LIN {X 0,Y 367.763,Z 472.156,A -85,B 0,C 180,E1 -12598.905,E2 -12598.905} C_VEL
LIN {X 0,Y 367.872,Z 472.925,A -85,B 0,C 180,E1 -12601.095,E2 -12601.095} C_VEL
LIN {X 0,Y 368.13,Z 472.594,A -85,B 0,C 180,E1 -12603.283,E2 -12603.283} C_VEL
LIN {X 0,Y 368.318,Z 471.288,A -85,B 0,C 180,E1 -12605.475,E2 -12605.475} C_VEL
LIN {X 0,Y 368.311,Z 470.292,A -85,B 0,C 180,E1 -12606.574,E2 -12606.574} C_VEL
LIN {X 0,Y 368.949,Z 467.35,A -85,B 0,C 180,E1 -12608.765,E2 -12608.765} C_VEL
LIN {X 0,Y 369.704,Z 463.365,A -85,B 0,C 180,E1 -12610.958,E2 -12610.958} C_VEL
LIN {X 0,Y 370.548,Z 458.282,A -85,B 0,C 180,E1 -12613.156,E2 -12613.156} C_VEL
LIN {X 0,Y 371.827,Z 451.616,A -85,B 0,C 180,E1 -12615.426,E2 -12615.426} C_VEL
LIN {X 0,Y 373.279,Z 444.114,A -85,B 0,C 180,E1 -12617.532,E2 -12617.532} C_VEL
LIN {X 0,Y 375.138,Z 434.807,A -85,B 0,C 180,E1 -12619.707,E2 -12619.707} C_VEL
LIN {X 0,Y 377.114,Z 425.21,A -85,B 0,C 180,E1 -12621.596,E2 -12621.596} C_VEL
LIN {X 0,Y 379.312,Z 413.922,A -85,B 0,C 180,E1 -12623.475,E2 -12623.475} C_VEL
LIN {X 0,Y 381.513,Z 402.619,A -85,B 0,C 180,E1 -12625.068,E2 -12625.068} C_VEL
LIN {X 0,Y 383.923,Z 389.529,A -85,B 0,C 180,E1 -12626.647,E2 -12626.647} C_VEL
LIN {X 0,Y 386.088,Z 376.887,A -85,B 0,C 180,E1 -12627.952,E2 -12627.952} C_VEL
LIN {X 0,Y 388.194,Z 363.605,A -85,B 0,C 180,E1 -12629.114,E2 -12629.114} C_VEL
LIN {X 0,Y 390.459,Z 347.831,A -85,B 0,C 180,E1 -12630.264,E2 -12630.264} C_VEL
LIN {X 0,Y 392.54,Z 330.694,A -85,B 0,C 180,E1 -12631.279,E2 -12631.279} C_VEL
LIN {X 0,Y 394.4,Z 312.888,A -85,B 0,C 180,E1 -12632.089,E2 -12632.089} C_VEL
LIN {X 0,Y 396.951,Z 285.614,A -85,B 0,C 180,E1 -12632.985,E2 -12632.985} C_VEL
LIN {X 0,Y 404.321,Z 221.247,A -85,B 0,C 180,E1 -12635.04,E2 -12635.04} C_VEL
LIN {X 0,Y 411.797,Z 167.375,A -85,B 0,C 180,E1 -12636.792,E2 -12636.792} C_VEL
LIN {X 0,Y 409.225,Z 162.785,A -85,B 0,C 180,E1 -12637.954,E2 -12637.954} C_VEL
LIN {X 0,Y 406.549,Z 158.694,A -85,B 0,C 180,E1 -12639.413,E2 -12639.413} C_VEL
LIN {X 0,Y 403.9,Z 155.628,A -85,B 0,C 180,E1 -12641.392,E2 -12641.392} C_VEL
LIN {X 0,Y 403.16,Z 154.958,A -85,B 0,C 180,E1 -12642.248,E2 -12642.248} C_VEL
LIN {X 0,Y 402.329,Z 154.997,A -85,B 0,C 180,E1 -12643.844,E2 -12643.844} C_VEL
LIN {X 0,Y 402.381,Z 156.776,A -85,B 0,C 180,E1 -12645.734,E2 -12645.734} C_VEL
LIN {X 0,Y 403.284,Z 159.225,A -85,B 0,C 180,E1 -12647.232,E2 -12647.232} C_VEL
LIN {X 0,Y 404.582,Z 162.984,A -85,B 0,C 180,E1 -12648.582,E2 -12648.582} C_VEL
LIN {X 0,Y 406.534,Z 167.981,A -85,B 0,C 180,E1 -12649.976,E2 -12649.976} C_VEL
LIN {X 0,Y 408.747,Z 174.299,A -85,B 0,C 180,E1 -12651.27,E2 -12651.27} C_VEL
LIN {X 0,Y 409.591,Z 177.225,A -85,B 0,C 180,E1 -12651.738,E2 -12651.738} C_VEL
LIN {X 0,Y 409.008,Z 196.365,A -85,B 0,C 180,E1 -12652.915,E2 -12652.915} C_VEL
LIN {X 0,Y 401.408,Z 257.244,A -85,B 0,C 180,E1 -12654.859,E2 -12654.859} C_VEL
LIN {X 0,Y 394.781,Z 323.074,A -85,B 0,C 180,E1 -12656.91,E2 -12656.91} C_VEL
LIN {X 0,Y 392.088,Z 351.319,A -85,B 0,C 180,E1 -12657.812,E2 -12657.812} C_VEL
LIN {X 0,Y 389.573,Z 370.272,A -85,B 0,C 180,E1 -12658.606,E2 -12658.606} C_VEL
LIN {X 0,Y 387.34,Z 385.034,A -85,B 0,C 180,E1 -12659.391,E2 -12659.391} C_VEL
LIN {X 0,Y 384.488,Z 402.958,A -85,B 0,C 180,E1 -12660.577,E2 -12660.577} C_VEL
LIN {X 0,Y 381.88,Z 418.792,A -85,B 0,C 180,E1 -12661.862,E2 -12661.862} C_VEL
LIN {X 0,Y 379.221,Z 433.932,A -85,B 0,C 180,E1 -12663.319,E2 -12663.319} C_VEL
LIN {X 0,Y 376.682,Z 448.794,A -85,B 0,C 180,E1 -12665.03,E2 -12665.03} C_VEL
LIN {X 0,Y 374.432,Z 462.363,A -85,B 0,C 180,E1 -12666.884,E2 -12666.884} C_VEL
LIN {X 0,Y 372.559,Z 473.762,A -85,B 0,C 180,E1 -12668.707,E2 -12668.707} C_VEL
LIN {X 0,Y 370.81,Z 485.557,A -85,B 0,C 180,E1 -12670.916,E2 -12670.916} C_VEL
LIN {X 0,Y 369.526,Z 495.557,A -85,B 0,C 180,E1 -12673.139,E2 -12673.139} C_VEL
LIN {X 0,Y 368.683,Z 503.018,A -85,B 0,C 180,E1 -12675.087,E2 -12675.087} C_VEL
LIN {X 0,Y 368.088,Z 510.152,A -85,B 0,C 180,E1 -12677.315,E2 -12677.315} C_VEL
LIN {X 0,Y 367.701,Z 516.033,A -85,B 0,C 180,E1 -12679.538,E2 -12679.538} C_VEL
LIN {X 0,Y 367.598,Z 520.659,A -85,B 0,C 180,E1 -12681.755,E2 -12681.755} C_VEL
LIN {X 0,Y 367.722,Z 523.703,A -85,B 0,C 180,E1 -12683.633,E2 -12683.633} C_VEL
LIN {X 0,Y 367.603,Z 525.957,A -85,B 0,C 180,E1 -12685.613,E2 -12685.613} C_VEL
LIN {X 0,Y 367.759,Z 527.494,A -85,B 0,C 180,E1 -12687.809,E2 -12687.809} C_VEL
LIN {X 0,Y 367.812,Z 527.835,A -85,B 0,C 180,E1 -12689.999,E2 -12689.999} C_VEL
LIN {X 0,Y 367.777,Z 527.091,A -85,B 0,C 180,E1 -12692.19,E2 -12692.19} C_VEL
LIN {X 0,Y 367.764,Z 526.32,A -85,B 0,C 180,E1 -12693.286,E2 -12693.286} C_VEL
LIN {X 0,Y 367.724,Z 523.809,A -85,B 0,C 180,E1 -12695.483,E2 -12695.483} C_VEL
LIN {X 0,Y 367.682,Z 520.167,A -85,B 0,C 180,E1 -12697.689,E2 -12697.689} C_VEL
LIN {X 0,Y 367.668,Z 515.275,A -85,B 0,C 180,E1 -12699.905,E2 -12699.905} C_VEL
LIN {X 0,Y 367.978,Z 509.03,A -85,B 0,C 180,E1 -12702.127,E2 -12702.127} C_VEL
LIN {X 0,Y 368.449,Z 501.363,A -85,B 0,C 180,E1 -12704.357,E2 -12704.357} C_VEL
LIN {X 0,Y 369.148,Z 493.386,A -85,B 0,C 180,E1 -12706.308,E2 -12706.308} C_VEL
LIN {X 0,Y 370.131,Z 483.052,A -85,B 0,C 180,E1 -12708.427,E2 -12708.427} C_VEL
LIN {X 0,Y 371.25,Z 472.812,A -85,B 0,C 180,E1 -12710.211,E2 -12710.211} C_VEL
LIN {X 0,Y 372.828,Z 459.757,A -85,B 0,C 180,E1 -12712.148,E2 -12712.148} C_VEL
LIN {X 0,Y 374.395,Z 446.566,A -85,B 0,C 180,E1 -12713.802,E2 -12713.802} C_VEL
LIN {X 0,Y 376.106,Z 432.348,A -85,B 0,C 180,E1 -12715.305,E2 -12715.305} C_VEL
LIN {X 0,Y 377.884,Z 416.601,A -85,B 0,C 180,E1 -12716.688,E2 -12716.688} C_VEL
LIN {X 0,Y 379.684,Z 400.106,A -85,B 0,C 180,E1 -12717.863,E2 -12717.863} C_VEL
LIN {X 0,Y 381.204,Z 383.748,A -85,B 0,C 180,E1 -12718.792,E2 -12718.792} C_VEL
LIN {X 0,Y 382.585,Z 366.326,A -85,B 0,C 180,E1 -12719.545,E2 -12719.545} C_VEL
LIN {X 0,Y 383.648,Z 349.415,A -85,B 0,C 180,E1 -12720.059,E2 -12720.059} C_VEL
LIN {X 0,Y 390.23,Z 192.191,A -85,B 0,C 180,E1 -12723.84,E2 -12723.84} C_VEL
LIN {X 0,Y 386.053,Z 158.999,A -85,B 0,C 180,E1 -12725.094,E2 -12725.094} C_VEL
LIN {X 0,Y 380.743,Z 146.981,A -85,B 0,C 180,E1 -12725.89,E2 -12725.89} C_VEL
LIN {X 0,Y 373.264,Z 123.838,A -85,B 0,C 180,E1 -12729.469,E2 -12729.469} C_VEL
LIN {X 0,Y 368.96,Z 110.84,A -85,B 0,C 180,E1 -12731.621,E2 -12731.621} C_VEL
LIN {X 0,Y 368.919,Z 110.844,A -85,B 0,C 180,E1 -12735.182,E2 -12735.182} C_VEL
LIN {X 0,Y 368.879,Z 110.849,A -85,B 0,C 180,E1 -12738.177,E2 -12738.177} C_VEL
LIN {X 0,Y 368.905,Z 110.841,A -85,B 0,C 180,E1 -12741.359,E2 -12741.359} C_VEL
LIN {X 0,Y 368.932,Z 110.838,A -85,B 0,C 180,E1 -12745.146,E2 -12745.146} C_VEL
LIN {X 0,Y 368.924,Z 110.839,A -85,B 0,C 180,E1 -12749.046,E2 -12749.046} C_VEL
LIN {X 0,Y 368.982,Z 110.833,A -85,B 0,C 180,E1 -12751.564,E2 -12751.564} C_VEL
LIN {X 0,Y 368.953,Z 110.836,A -85,B 0,C 180,E1 -12755.224,E2 -12755.224} C_VEL
LIN {X 0,Y 368.932,Z 110.838,A -85,B 0,C 180,E1 -12758.973,E2 -12758.973} C_VEL
LIN {X 0,Y 368.986,Z 110.834,A -85,B 0,C 180,E1 -12762.257,E2 -12762.257} C_VEL
LIN {X 0,Y 369.012,Z 110.832,A -85,B 0,C 180,E1 -12765.665,E2 -12765.665} C_VEL
LIN {X 0,Y 369.025,Z 110.827,A -85,B 0,C 180,E1 -12769.021,E2 -12769.021} C_VEL
LIN {X 0,Y 369.183,Z 110.808,A -85,B 0,C 180,E1 -12772.342,E2 -12772.342} C_VEL
LIN {X 0,Y 369.14,Z 110.812,A -85,B 0,C 180,E1 -12774.538,E2 -12774.538} C_VEL
LIN {X 0,Y 369.314,Z 110.795,A -85,B 0,C 180,E1 -12777.819,E2 -12777.819} C_VEL
LIN {X 0,Y 369.454,Z 110.776,A -85,B 0,C 180,E1 -12780,E2 -12780} C_VEL
LIN {X 0,Y 369.314,Z 110.792,A -85,B 0,C 180,E1 -12782.181,E2 -12782.181} C_VEL
LIN {X 0,Y 369.2,Z 110.805,A -85,B 0,C 180,E1 -12786.616,E2 -12786.616} C_VEL
LIN {X 0,Y 369.133,Z 110.814,A -85,B 0,C 180,E1 -12788.761,E2 -12788.761} C_VEL
LIN {X 0,Y 369.001,Z 110.83,A -85,B 0,C 180,E1 -12792.094,E2 -12792.094} C_VEL
LIN {X 0,Y 368.993,Z 110.836,A -85,B 0,C 180,E1 -12795.465,E2 -12795.465} C_VEL
LIN {X 0,Y 368.954,Z 110.838,A -85,B 0,C 180,E1 -12798.894,E2 -12798.894} C_VEL
LIN {X 0,Y 368.928,Z 110.839,A -85,B 0,C 180,E1 -12802.395,E2 -12802.395} C_VEL
LIN {X 0,Y 368.996,Z 110.83,A -85,B 0,C 180,E1 -12805.981,E2 -12805.981} C_VEL
LIN {X 0,Y 368.911,Z 110.842,A -85,B 0,C 180,E1 -12809.691,E2 -12809.691} C_VEL
LIN {X 0,Y 368.893,Z 110.85,A -85,B 0,C 180,E1 -12813.044,E2 -12813.044} C_VEL
LIN {X 0,Y 368.914,Z 110.841,A -85,B 0,C 180,E1 -12816.197,E2 -12816.197} C_VEL
LIN {X 0,Y 368.901,Z 110.849,A -85,B 0,C 180,E1 -12818.953,E2 -12818.953} C_VEL
LIN {X 0,Y 368.878,Z 110.845,A -85,B 0,C 180,E1 -12822.01,E2 -12822.01} C_VEL
LIN {X 0,Y 368.905,Z 110.844,A -85,B 0,C 180,E1 -12825.181,E2 -12825.181} C_VEL
LIN {X 0,Y 368.907,Z 110.842,A -85,B 0,C 180,E1 -12828.182,E2 -12828.182} C_VEL
LIN {X 0,Y 368.908,Z 110.842,A -85,B 0,C 180,E1 -12831.36,E2 -12831.36} C_VEL
LIN {X 0,Y 368.934,Z 110.84,A -85,B 0,C 180,E1 -12835.147,E2 -12835.147} C_VEL
LIN {X 0,Y 368.927,Z 110.841,A -85,B 0,C 180,E1 -12839.047,E2 -12839.047} C_VEL
LIN {X 0,Y 368.961,Z 110.838,A -85,B 0,C 180,E1 -12842.797,E2 -12842.797} C_VEL
LIN {X 0,Y 368.944,Z 110.839,A -85,B 0,C 180,E1 -12846.114,E2 -12846.114} C_VEL
LIN {X 0,Y 368.944,Z 110.839,A -85,B 0,C 180,E1 -12849.948,E2 -12849.948} C_VEL
LIN {X 0,Y 368.975,Z 110.833,A -85,B 0,C 180,E1 -12853.399,E2 -12853.399} C_VEL
LIN {X 0,Y 369.057,Z 110.824,A -85,B 0,C 180,E1 -12856.791,E2 -12856.791} C_VEL
LIN {X 0,Y 369.07,Z 110.826,A -85,B 0,C 180,E1 -12860.133,E2 -12860.133} C_VEL
LIN {X 0,Y 369.189,Z 110.811,A -85,B 0,C 180,E1 -12862.343,E2 -12862.343} C_VEL
LIN {X 0,Y 369.144,Z 110.814,A -85,B 0,C 180,E1 -12864.538,E2 -12864.538} C_VEL
LIN {X 0,Y 369.317,Z 110.794,A -85,B 0,C 180,E1 -12867.82,E2 -12867.82} C_VEL
LIN {X 0,Y 369.457,Z 110.779,A -85,B 0,C 180,E1 -12870.001,E2 -12870.001} C_VEL
LIN {X 0,Y 369.317,Z 110.795,A -85,B 0,C 180,E1 -12872.182,E2 -12872.182} C_VEL
LIN {X 0,Y 369.21,Z 110.805,A -85,B 0,C 180,E1 -12876.559,E2 -12876.559} C_VEL
LIN {X 0,Y 369.139,Z 110.812,A -85,B 0,C 180,E1 -12878.762,E2 -12878.762} C_VEL
LIN {X 0,Y 369.007,Z 110.833,A -85,B 0,C 180,E1 -12882.094,E2 -12882.094} C_VEL
LIN {X 0,Y 369,Z 110.833,A -85,B 0,C 180,E1 -12885.465,E2 -12885.465} C_VEL
LIN {X 0,Y 368.96,Z 110.835,A -85,B 0,C 180,E1 -12888.895,E2 -12888.895} C_VEL
LIN {X 0,Y 368.934,Z 110.838,A -85,B 0,C 180,E1 -12892.396,E2 -12892.396} C_VEL
LIN {X 0,Y 369.002,Z 110.832,A -85,B 0,C 180,E1 -12895.981,E2 -12895.981} C_VEL
LIN {X 0,Y 368.917,Z 110.845,A -85,B 0,C 180,E1 -12899.691,E2 -12899.691} C_VEL
LIN {X 0,Y 368.899,Z 110.844,A -85,B 0,C 180,E1 -12903.044,E2 -12903.044} C_VEL
LIN {X 0,Y 368.92,Z 110.84,A -85,B 0,C 180,E1 -12906.197,E2 -12906.197} C_VEL
LIN {X 0,Y 368.906,Z 110.844,A -85,B 0,C 180,E1 -12908.954,E2 -12908.954} C_VEL
LIN {X 0,Y 368.885,Z 110.845,A -85,B 0,C 180,E1 -12912.01,E2 -12912.01} C_VEL
LIN {X 0,Y 368.885,Z 110.846,A -85,B 0,C 180,E1 -12914.768,E2 -12914.768} C_VEL
LIN {X 0,Y 368.259,Z 110.929,A -85,B 0,C 180,E1 -12915.679,E2 -12915.679} C_VEL
LIN {X 0,Y 365.4,Z 111.29,A -85,B 0,C 180,E1 -12917.16,E2 -12917.16} C_VEL
LIN {X 0,Y 362.957,Z 111.592,A -85,B 0,C 180,E1 -12918.358,E2 -12918.358} C_VEL
LIN {X 0,Y 361.915,Z 111.718,A -85,B 0,C 180,E1 -12919.286,E2 -12919.286} C_VEL
LIN {X 0,Y 361.836,Z 111.724,A -85,B 0,C 180,E1 -12919.6,E2 -12919.6} C_VEL
LIN {X 0,Y 361.894,Z 111.804,A -85,B 0,C 180,E1 -12923.315,E2 -12923.315} C_VEL
LIN {X 0,Y 362.879,Z 114.579,A -85,B 0,C 180,E1 -12923.489,E2 -12923.489} C_VEL
LIN {X 0,Y 375.869,Z 139.954,A -85,B 0,C 180,E1 -12925.358,E2 -12925.358} C_VEL
LIN {X 0,Y 383.362,Z 155.105,A -85,B 0,C 180,E1 -12926.389,E2 -12926.389} C_VEL
LIN {X 0,Y 377.045,Z 300.554,A -85,B 0,C 180,E1 -12929.976,E2 -12929.976} C_VEL
LIN {X 0,Y 376.115,Z 317.935,A -85,B 0,C 180,E1 -12930.626,E2 -12930.626} C_VEL
LIN {X 0,Y 374.874,Z 335.248,A -85,B 0,C 180,E1 -12931.502,E2 -12931.502} C_VEL
LIN {X 0,Y 373.524,Z 351.415,A -85,B 0,C 180,E1 -12932.55,E2 -12932.55} C_VEL
LIN {X 0,Y 371.952,Z 367.033,A -85,B 0,C 180,E1 -12933.79,E2 -12933.79} C_VEL
LIN {X 0,Y 370.293,Z 381.51,A -85,B 0,C 180,E1 -12935.17,E2 -12935.17} C_VEL
LIN {X 0,Y 368.602,Z 396.146,A -85,B 0,C 180,E1 -12936.843,E2 -12936.843} C_VEL
LIN {X 0,Y 367.227,Z 407.642,A -85,B 0,C 180,E1 -12938.383,E2 -12938.383} C_VEL
LIN {X 0,Y 365.713,Z 420.041,A -85,B 0,C 180,E1 -12940.331,E2 -12940.331} C_VEL
LIN {X 0,Y 364.399,Z 430.687,A -85,B 0,C 180,E1 -12942.316,E2 -12942.316} C_VEL
LIN {X 0,Y 363.327,Z 439.7,A -85,B 0,C 180,E1 -12944.288,E2 -12944.288} C_VEL
LIN {X 0,Y 362.42,Z 448.408,A -85,B 0,C 180,E1 -12946.544,E2 -12946.544} C_VEL
LIN {X 0,Y 361.695,Z 455.627,A -85,B 0,C 180,E1 -12948.796,E2 -12948.796} C_VEL
LIN {X 0,Y 361.288,Z 461.435,A -85,B 0,C 180,E1 -12951.047,E2 -12951.047} C_VEL
LIN {X 0,Y 361.011,Z 466.025,A -85,B 0,C 180,E1 -12953.292,E2 -12953.292} C_VEL
LIN {X 0,Y 360.792,Z 469.537,A -85,B 0,C 180,E1 -12955.531,E2 -12955.531} C_VEL
LIN {X 0,Y 360.773,Z 471.872,A -85,B 0,C 180,E1 -12957.767,E2 -12957.767} C_VEL
LIN {X 0,Y 360.743,Z 473.22,A -85,B 0,C 180,E1 -12960,E2 -12960} C_VEL
LIN {X 0,Y 360.957,Z 473.516,A -85,B 0,C 180,E1 -12962.232,E2 -12962.232} C_VEL
LIN {X 0,Y 361.142,Z 472.773,A -85,B 0,C 180,E1 -12964.464,E2 -12964.464} C_VEL
LIN {X 0,Y 361.296,Z 471.082,A -85,B 0,C 180,E1 -12966.702,E2 -12966.702} C_VEL
LIN {X 0,Y 361.982,Z 468.215,A -85,B 0,C 180,E1 -12968.935,E2 -12968.935} C_VEL
LIN {X 0,Y 362.787,Z 464.338,A -85,B 0,C 180,E1 -12971.17,E2 -12971.17} C_VEL
LIN {X 0,Y 363.683,Z 459.323,A -85,B 0,C 180,E1 -12973.408,E2 -12973.408} C_VEL
LIN {X 0,Y 365.063,Z 452.768,A -85,B 0,C 180,E1 -12975.723,E2 -12975.723} C_VEL
LIN {X 0,Y 366.634,Z 445.41,A -85,B 0,C 180,E1 -12977.861,E2 -12977.861} C_VEL
LIN {X 0,Y 368.616,Z 436.268,A -85,B 0,C 180,E1 -12980.071,E2 -12980.071} C_VEL
LIN {X 0,Y 371.062,Z 425.321,A -85,B 0,C 180,E1 -12982.259,E2 -12982.259} C_VEL
LIN {X 0,Y 373.402,Z 414.056,A -85,B 0,C 180,E1 -12984.165,E2 -12984.165} C_VEL
LIN {X 0,Y 375.766,Z 402.839,A -85,B 0,C 180,E1 -12985.757,E2 -12985.757} C_VEL
LIN {X 0,Y 378.539,Z 388.47,A -85,B 0,C 180,E1 -12987.505,E2 -12987.505} C_VEL
LIN {X 0,Y 381.359,Z 372.824,A -85,B 0,C 180,E1 -12989.082,E2 -12989.082} C_VEL
LIN {X 0,Y 384.215,Z 355.813,A -85,B 0,C 180,E1 -12990.474,E2 -12990.474} C_VEL
LIN {X 0,Y 386.746,Z 338.182,A -85,B 0,C 180,E1 -12991.634,E2 -12991.634} C_VEL
LIN {X 0,Y 388.751,Z 321.708,A -85,B 0,C 180,E1 -12992.498,E2 -12992.498} C_VEL
LIN {X 0,Y 390.581,Z 303.73,A -85,B 0,C 180,E1 -12993.208,E2 -12993.208} C_VEL
LIN {X 0,Y 397.716,Z 242.686,A -85,B 0,C 180,E1 -12995.198,E2 -12995.198} C_VEL
LIN {X 0,Y 408.086,Z 171.591,A -85,B 0,C 180,E1 -12997.562,E2 -12997.562} C_VEL
LIN {X 0,Y 406.02,Z 168.026,A -85,B 0,C 180,E1 -12998.612,E2 -12998.612} C_VEL
LIN {X 0,Y 404.236,Z 165.141,A -85,B 0,C 180,E1 -12999.709,E2 -12999.709} C_VEL
LIN {X 0,Y 402.038,Z 162.435,A -85,B 0,C 180,E1 -13001.503,E2 -13001.503} C_VEL
LIN {X 0,Y 401.149,Z 161.75,A -85,B 0,C 180,E1 -13002.622,E2 -13002.622} C_VEL
LIN {X 0,Y 400.531,Z 162.015,A -85,B 0,C 180,E1 -13003.993,E2 -13003.993} C_VEL
LIN {X 0,Y 400.659,Z 163.827,A -85,B 0,C 180,E1 -13005.822,E2 -13005.822} C_VEL
LIN {X 0,Y 401.583,Z 166.692,A -85,B 0,C 180,E1 -13007.371,E2 -13007.371} C_VEL
LIN {X 0,Y 403.632,Z 172.828,A -85,B 0,C 180,E1 -13009.313,E2 -13009.313} C_VEL
LIN {X 0,Y 405.733,Z 179.636,A -85,B 0,C 180,E1 -13010.767,E2 -13010.767} C_VEL
LIN {X 0,Y 406.152,Z 181.286,A -85,B 0,C 180,E1 -13011.038,E2 -13011.038} C_VEL
LIN {X 0,Y 405.317,Z 198.198,A -85,B 0,C 180,E1 -13012.103,E2 -13012.103} C_VEL
LIN {X 0,Y 396.177,Z 266.329,A -85,B 0,C 180,E1 -13014.324,E2 -13014.324} C_VEL
LIN {X 0,Y 389.101,Z 332.133,A -85,B 0,C 180,E1 -13016.424,E2 -13016.424} C_VEL
LIN {X 0,Y 386.846,Z 352.633,A -85,B 0,C 180,E1 -13017.128,E2 -13017.128} C_VEL
LIN {X 0,Y 384.101,Z 371.38,A -85,B 0,C 180,E1 -13017.952,E2 -13017.952} C_VEL
LIN {X 0,Y 381.631,Z 386.548,A -85,B 0,C 180,E1 -13018.805,E2 -13018.805} C_VEL
LIN {X 0,Y 378.451,Z 404.704,A -85,B 0,C 180,E1 -13020.06,E2 -13020.06} C_VEL
LIN {X 0,Y 375.719,Z 419.977,A -85,B 0,C 180,E1 -13021.358,E2 -13021.358} C_VEL
LIN {X 0,Y 372.732,Z 435.816,A -85,B 0,C 180,E1 -13022.958,E2 -13022.958} C_VEL
LIN {X 0,Y 370.057,Z 450.273,A -85,B 0,C 180,E1 -13024.702,E2 -13024.702} C_VEL
LIN {X 0,Y 367.778,Z 463.128,A -85,B 0,C 180,E1 -13026.527,E2 -13026.527} C_VEL
LIN {X 0,Y 365.886,Z 473.862,A -85,B 0,C 180,E1 -13028.299,E2 -13028.299} C_VEL
LIN {X 0,Y 364.173,Z 484.144,A -85,B 0,C 180,E1 -13030.261,E2 -13030.261} C_VEL
LIN {X 0,Y 362.743,Z 494.248,A -85,B 0,C 180,E1 -13032.523,E2 -13032.523} C_VEL
LIN {X 0,Y 361.685,Z 502.788,A -85,B 0,C 180,E1 -13034.791,E2 -13034.791} C_VEL
LIN {X 0,Y 361.047,Z 510.035,A -85,B 0,C 180,E1 -13037.134,E2 -13037.134} C_VEL
LIN {X 0,Y 360.623,Z 515.639,A -85,B 0,C 180,E1 -13039.33,E2 -13039.33} C_VEL
LIN {X 0,Y 360.519,Z 520.243,A -85,B 0,C 180,E1 -13041.592,E2 -13041.592} C_VEL
LIN {X 0,Y 360.644,Z 523.385,A -85,B 0,C 180,E1 -13043.642,E2 -13043.642} C_VEL
LIN {X 0,Y 360.532,Z 525.452,A -85,B 0,C 180,E1 -13045.527,E2 -13045.527} C_VEL
LIN {X 0,Y 360.691,Z 526.924,A -85,B 0,C 180,E1 -13047.766,E2 -13047.766} C_VEL
LIN {X 0,Y 360.765,Z 527.242,A -85,B 0,C 180,E1 -13049.999,E2 -13049.999} C_VEL
LIN {X 0,Y 360.711,Z 526.425,A -85,B 0,C 180,E1 -13052.232,E2 -13052.232} C_VEL
LIN {X 0,Y 360.557,Z 524.488,A -85,B 0,C 180,E1 -13054.471,E2 -13054.471} C_VEL
LIN {X 0,Y 360.695,Z 521.812,A -85,B 0,C 180,E1 -13056.43,E2 -13056.43} C_VEL
LIN {X 0,Y 360.595,Z 517.008,A -85,B 0,C 180,E1 -13058.969,E2 -13058.969} C_VEL
LIN {X 0,Y 360.754,Z 511.368,A -85,B 0,C 180,E1 -13061.233,E2 -13061.233} C_VEL
LIN {X 0,Y 361.178,Z 504.313,A -85,B 0,C 180,E1 -13063.503,E2 -13063.503} C_VEL
LIN {X 0,Y 361.821,Z 495.725,A -85,B 0,C 180,E1 -13065.779,E2 -13065.779} C_VEL
LIN {X 0,Y 362.713,Z 486.824,A -85,B 0,C 180,E1 -13067.768,E2 -13067.768} C_VEL
LIN {X 0,Y 363.81,Z 476.313,A -85,B 0,C 180,E1 -13069.758,E2 -13069.758} C_VEL
LIN {X 0,Y 365.307,Z 463.947,A -85,B 0,C 180,E1 -13071.736,E2 -13071.736} C_VEL
LIN {X 0,Y 366.89,Z 451.226,A -85,B 0,C 180,E1 -13073.458,E2 -13073.458} C_VEL
LIN {X 0,Y 368.615,Z 436.88,A -85,B 0,C 180,E1 -13075.1,E2 -13075.1} C_VEL
LIN {X 0,Y 370.387,Z 422.46,A -85,B 0,C 180,E1 -13076.48,E2 -13076.48} C_VEL
LIN {X 0,Y 372.178,Z 406.983,A -85,B 0,C 180,E1 -13077.709,E2 -13077.709} C_VEL
LIN {X 0,Y 373.777,Z 391.291,A -85,B 0,C 180,E1 -13078.727,E2 -13078.727} C_VEL
LIN {X 0,Y 375.357,Z 374.103,A -85,B 0,C 180,E1 -13079.592,E2 -13079.592} C_VEL
LIN {X 0,Y 376.663,Z 356.279,A -85,B 0,C 180,E1 -13080.25,E2 -13080.25} C_VEL
LIN {X 0,Y 383.889,Z 193.183,A -85,B 0,C 180,E1 -13084.298,E2 -13084.298} C_VEL
LIN {X 0,Y 379.923,Z 161.529,A -85,B 0,C 180,E1 -13085.518,E2 -13085.518} C_VEL
LIN {X 0,Y 373.298,Z 146.581,A -85,B 0,C 180,E1 -13086.519,E2 -13086.519} C_VEL
LIN {X 0,Y 367.039,Z 127.165,A -85,B 0,C 180,E1 -13089.578,E2 -13089.578} C_VEL
LIN {X 0,Y 361.894,Z 111.721,A -85,B 0,C 180,E1 -13092.17,E2 -13092.17} C_VEL
LIN {X 0,Y 361.842,Z 111.726,A -85,B 0,C 180,E1 -13095.636,E2 -13095.636} C_VEL
LIN {X 0,Y 361.831,Z 111.723,A -85,B 0,C 180,E1 -13099.244,E2 -13099.244} C_VEL
LIN {X 0,Y 361.867,Z 111.72,A -85,B 0,C 180,E1 -13102.775,E2 -13102.775} C_VEL
LIN {X 0,Y 361.851,Z 111.722,A -85,B 0,C 180,E1 -13105.72,E2 -13105.72} C_VEL
LIN {X 0,Y 361.872,Z 111.719,A -85,B 0,C 180,E1 -13109.672,E2 -13109.672} C_VEL
LIN {X 0,Y 361.95,Z 111.709,A -85,B 0,C 180,E1 -13113.475,E2 -13113.475} C_VEL
LIN {X 0,Y 361.885,Z 111.716,A -85,B 0,C 180,E1 -13117.145,E2 -13117.145} C_VEL
LIN {X 0,Y 361.916,Z 111.712,A -85,B 0,C 180,E1 -13120.724,E2 -13120.724} C_VEL
LIN {X 0,Y 361.944,Z 111.712,A -85,B 0,C 180,E1 -13124.226,E2 -13124.226} C_VEL
LIN {X 0,Y 361.995,Z 111.703,A -85,B 0,C 180,E1 -13126.528,E2 -13126.528} C_VEL
LIN {X 0,Y 362.031,Z 111.703,A -85,B 0,C 180,E1 -13129.938,E2 -13129.938} C_VEL
LIN {X 0,Y 362.146,Z 111.686,A -85,B 0,C 180,E1 -13132.193,E2 -13132.193} C_VEL
LIN {X 0,Y 362.114,Z 111.688,A -85,B 0,C 180,E1 -13134.431,E2 -13134.431} C_VEL
LIN {X 0,Y 362.278,Z 111.672,A -85,B 0,C 180,E1 -13137.777,E2 -13137.777} C_VEL
LIN {X 0,Y 362.423,Z 111.652,A -85,B 0,C 180,E1 -13140,E2 -13140} C_VEL
LIN {X 0,Y 362.278,Z 111.668,A -85,B 0,C 180,E1 -13142.224,E2 -13142.224} C_VEL
LIN {X 0,Y 362.168,Z 111.681,A -85,B 0,C 180,E1 -13146.686,E2 -13146.686} C_VEL
LIN {X 0,Y 362.069,Z 111.694,A -85,B 0,C 180,E1 -13148.933,E2 -13148.933} C_VEL
LIN {X 0,Y 361.956,Z 111.707,A -85,B 0,C 180,E1 -13152.333,E2 -13152.333} C_VEL
LIN {X 0,Y 361.957,Z 111.707,A -85,B 0,C 180,E1 -13154.621,E2 -13154.621} C_VEL
LIN {X 0,Y 361.951,Z 111.708,A -85,B 0,C 180,E1 -13158.1,E2 -13158.1} C_VEL
LIN {X 0,Y 361.887,Z 111.718,A -85,B 0,C 180,E1 -13161.653,E2 -13161.653} C_VEL
LIN {X 0,Y 361.924,Z 111.716,A -85,B 0,C 180,E1 -13165.29,E2 -13165.29} C_VEL
LIN {X 0,Y 361.904,Z 111.714,A -85,B 0,C 180,E1 -13167.779,E2 -13167.779} C_VEL
LIN {X 0,Y 361.833,Z 111.724,A -85,B 0,C 180,E1 -13171.63,E2 -13171.63} C_VEL
LIN {X 0,Y 361.871,Z 111.721,A -85,B 0,C 180,E1 -13175.345,E2 -13175.345} C_VEL
LIN {X 0,Y 361.868,Z 111.724,A -85,B 0,C 180,E1 -13179.028,E2 -13179.028} C_VEL
LIN {X 0,Y 361.833,Z 111.728,A -85,B 0,C 180,E1 -13182.829,E2 -13182.829} C_VEL
LIN {X 0,Y 361.834,Z 111.722,A -85,B 0,C 180,E1 -13185.944,E2 -13185.944} C_VEL
LIN {X 0,Y 361.87,Z 111.72,A -85,B 0,C 180,E1 -13189.238,E2 -13189.238} C_VEL
LIN {X 0,Y 361.869,Z 111.721,A -85,B 0,C 180,E1 -13192.983,E2 -13192.983} C_VEL
LIN {X 0,Y 361.856,Z 111.726,A -85,B 0,C 180,E1 -13196.631,E2 -13196.631} C_VEL
LIN {X 0,Y 361.871,Z 111.718,A -85,B 0,C 180,E1 -13199.673,E2 -13199.673} C_VEL
LIN {X 0,Y 361.952,Z 111.708,A -85,B 0,C 180,E1 -13203.476,E2 -13203.476} C_VEL
LIN {X 0,Y 361.892,Z 111.716,A -85,B 0,C 180,E1 -13207.146,E2 -13207.146} C_VEL
LIN {X 0,Y 361.927,Z 111.714,A -85,B 0,C 180,E1 -13210.725,E2 -13210.725} C_VEL
LIN {X 0,Y 361.945,Z 111.714,A -85,B 0,C 180,E1 -13214.227,E2 -13214.227} C_VEL
LIN {X 0,Y 361.998,Z 111.706,A -85,B 0,C 180,E1 -13216.529,E2 -13216.529} C_VEL
LIN {X 0,Y 362.033,Z 111.701,A -85,B 0,C 180,E1 -13219.939,E2 -13219.939} C_VEL
LIN {X 0,Y 362.152,Z 111.689,A -85,B 0,C 180,E1 -13222.193,E2 -13222.193} C_VEL
LIN {X 0,Y 362.118,Z 111.69,A -85,B 0,C 180,E1 -13224.432,E2 -13224.432} C_VEL
LIN {X 0,Y 362.281,Z 111.67,A -85,B 0,C 180,E1 -13227.777,E2 -13227.777} C_VEL
LIN {X 0,Y 362.427,Z 111.654,A -85,B 0,C 180,E1 -13230.001,E2 -13230.001} C_VEL
LIN {X 0,Y 362.281,Z 111.671,A -85,B 0,C 180,E1 -13232.224,E2 -13232.224} C_VEL
LIN {X 0,Y 362.173,Z 111.68,A -85,B 0,C 180,E1 -13236.687,E2 -13236.687} C_VEL
LIN {X 0,Y 362.075,Z 111.692,A -85,B 0,C 180,E1 -13238.934,E2 -13238.934} C_VEL
LIN {X 0,Y 361.962,Z 111.708,A -85,B 0,C 180,E1 -13242.333,E2 -13242.333} C_VEL
LIN {X 0,Y 361.964,Z 111.706,A -85,B 0,C 180,E1 -13244.621,E2 -13244.621} C_VEL
LIN {X 0,Y 361.958,Z 111.71,A -85,B 0,C 180,E1 -13248.1,E2 -13248.1} C_VEL
LIN {X 0,Y 361.894,Z 111.721,A -85,B 0,C 180,E1 -13251.654,E2 -13251.654} C_VEL
LIN {X 0,Y 361.93,Z 111.713,A -85,B 0,C 180,E1 -13255.291,E2 -13255.291} C_VEL
LIN {X 0,Y 361.911,Z 111.717,A -85,B 0,C 180,E1 -13257.78,E2 -13257.78} C_VEL
LIN {X 0,Y 361.84,Z 111.727,A -85,B 0,C 180,E1 -13261.63,E2 -13261.63} C_VEL
LIN {X 0,Y 361.877,Z 111.722,A -85,B 0,C 180,E1 -13265.345,E2 -13265.345} C_VEL
LIN {X 0,Y 361.872,Z 111.72,A -85,B 0,C 180,E1 -13269.027,E2 -13269.027} C_VEL
LIN {X 0,Y 361.84,Z 111.723,A -85,B 0,C 180,E1 -13272.829,E2 -13272.829} C_VEL
LIN {X 0,Y 361.838,Z 111.722,A -85,B 0,C 180,E1 -13275.944,E2 -13275.944} C_VEL
LIN {X 0,Y 361.836,Z 111.724,A -85,B 0,C 180,E1 -13279.6,E2 -13279.6} C_VEL
LIN {X 0,Y 361.126,Z 111.811,A -85,B 0,C 180,E1 -13279.96,E2 -13279.96} C_VEL
LIN {X 0,Y 355.306,Z 112.541,A -85,B 0,C 180,E1 -13281.011,E2 -13281.011} C_VEL
LIN {X 0,Y 354.786,Z 112.598,A -85,B 0,C 180,E1 -13281.324,E2 -13281.324} C_VEL
LIN {X 0,Y 354.847,Z 112.799,A -85,B 0,C 180,E1 -13282.701,E2 -13282.701} C_VEL
LIN {X 0,Y 356.002,Z 115.688,A -85,B 0,C 180,E1 -13282.9,E2 -13282.9} C_VEL
LIN {X 0,Y 370.222,Z 143.551,A -85,B 0,C 180,E1 -13285.004,E2 -13285.004} C_VEL
LIN {X 0,Y 376.96,Z 157.248,A -85,B 0,C 180,E1 -13285.95,E2 -13285.95} C_VEL
LIN {X 0,Y 370.457,Z 300.822,A -85,B 0,C 180,E1 -13289.583,E2 -13289.583} C_VEL
LIN {X 0,Y 369.485,Z 318.162,A -85,B 0,C 180,E1 -13290.242,E2 -13290.242} C_VEL
LIN {X 0,Y 368.245,Z 335.127,A -85,B 0,C 180,E1 -13291.112,E2 -13291.112} C_VEL
LIN {X 0,Y 366.945,Z 350.322,A -85,B 0,C 180,E1 -13292.101,E2 -13292.101} C_VEL
LIN {X 0,Y 365.431,Z 365.345,A -85,B 0,C 180,E1 -13293.285,E2 -13293.285} C_VEL
LIN {X 0,Y 363.737,Z 380.208,A -85,B 0,C 180,E1 -13294.691,E2 -13294.691} C_VEL
LIN {X 0,Y 362.07,Z 394.03,A -85,B 0,C 180,E1 -13296.248,E2 -13296.248} C_VEL
LIN {X 0,Y 360.488,Z 406.842,A -85,B 0,C 180,E1 -13297.957,E2 -13297.957} C_VEL
LIN {X 0,Y 358.918,Z 418.788,A -85,B 0,C 180,E1 -13299.832,E2 -13299.832} C_VEL
LIN {X 0,Y 357.759,Z 428.842,A -85,B 0,C 180,E1 -13301.681,E2 -13301.681} C_VEL
LIN {X 0,Y 356.561,Z 438.278,A -85,B 0,C 180,E1 -13303.688,E2 -13303.688} C_VEL
LIN {X 0,Y 355.603,Z 447.27,A -85,B 0,C 180,E1 -13305.967,E2 -13305.967} C_VEL
LIN {X 0,Y 354.858,Z 453.941,A -85,B 0,C 180,E1 -13307.997,E2 -13307.997} C_VEL
LIN {X 0,Y 354.354,Z 460.237,A -85,B 0,C 180,E1 -13310.294,E2 -13310.294} C_VEL
LIN {X 0,Y 354.023,Z 465.268,A -85,B 0,C 180,E1 -13312.587,E2 -13312.587} C_VEL
LIN {X 0,Y 353.824,Z 468.249,A -85,B 0,C 180,E1 -13314.3,E2 -13314.3} C_VEL
LIN {X 0,Y 353.768,Z 471.232,A -85,B 0,C 180,E1 -13316.583,E2 -13316.583} C_VEL
LIN {X 0,Y 353.622,Z 473.177,A -85,B 0,C 180,E1 -13318.861,E2 -13318.861} C_VEL
LIN {X 0,Y 353.752,Z 474.106,A -85,B 0,C 180,E1 -13321.138,E2 -13321.138} C_VEL
LIN {X 0,Y 354.006,Z 473.932,A -85,B 0,C 180,E1 -13323.414,E2 -13323.414} C_VEL
LIN {X 0,Y 354.247,Z 472.824,A -85,B 0,C 180,E1 -13325.693,E2 -13325.693} C_VEL
LIN {X 0,Y 354.691,Z 470.601,A -85,B 0,C 180,E1 -13327.973,E2 -13327.973} C_VEL
LIN {X 0,Y 355.632,Z 466.363,A -85,B 0,C 180,E1 -13330.821,E2 -13330.821} C_VEL
LIN {X 0,Y 356.576,Z 461.736,A -85,B 0,C 180,E1 -13333.1,E2 -13333.1} C_VEL
LIN {X 0,Y 357.768,Z 456.341,A -85,B 0,C 180,E1 -13335.228,E2 -13335.228} C_VEL
LIN {X 0,Y 359.499,Z 448.77,A -85,B 0,C 180,E1 -13337.639,E2 -13337.639} C_VEL
LIN {X 0,Y 361.504,Z 440.165,A -85,B 0,C 180,E1 -13339.89,E2 -13339.89} C_VEL
LIN {X 0,Y 363.891,Z 430.37,A -85,B 0,C 180,E1 -13342.019,E2 -13342.019} C_VEL
LIN {X 0,Y 366.426,Z 419.315,A -85,B 0,C 180,E1 -13344.052,E2 -13344.052} C_VEL
LIN {X 0,Y 368.793,Z 408.856,A -85,B 0,C 180,E1 -13345.692,E2 -13345.692} C_VEL
LIN {X 0,Y 371.968,Z 394.556,A -85,B 0,C 180,E1 -13347.574,E2 -13347.574} C_VEL
LIN {X 0,Y 374.384,Z 382.571,A -85,B 0,C 180,E1 -13348.906,E2 -13348.906} C_VEL
LIN {X 0,Y 376.963,Z 368.803,A -85,B 0,C 180,E1 -13350.224,E2 -13350.224} C_VEL
LIN {X 0,Y 379.87,Z 352.083,A -85,B 0,C 180,E1 -13351.54,E2 -13351.54} C_VEL
LIN {X 0,Y 382.336,Z 335.545,A -85,B 0,C 180,E1 -13352.603,E2 -13352.603} C_VEL
LIN {X 0,Y 384.612,Z 318.095,A -85,B 0,C 180,E1 -13353.478,E2 -13353.478} C_VEL
LIN {X 0,Y 387.219,Z 294.469,A -85,B 0,C 180,E1 -13354.357,E2 -13354.357} C_VEL
LIN {X 0,Y 395.294,Z 234.204,A -85,B 0,C 180,E1 -13356.378,E2 -13356.378} C_VEL
LIN {X 0,Y 404.599,Z 176.2,A -85,B 0,C 180,E1 -13358.332,E2 -13358.332} C_VEL
LIN {X 0,Y 402.314,Z 171.99,A -85,B 0,C 180,E1 -13359.768,E2 -13359.768} C_VEL
LIN {X 0,Y 400.053,Z 169.129,A -85,B 0,C 180,E1 -13361.713,E2 -13361.713} C_VEL
LIN {X 0,Y 399.544,Z 168.662,A -85,B 0,C 180,E1 -13362.371,E2 -13362.371} C_VEL
LIN {X 0,Y 398.853,Z 168.739,A -85,B 0,C 180,E1 -13363.743,E2 -13363.743} C_VEL
LIN {X 0,Y 398.82,Z 170.592,A -85,B 0,C 180,E1 -13365.669,E2 -13365.669} C_VEL
LIN {X 0,Y 399.533,Z 173.241,A -85,B 0,C 180,E1 -13367.108,E2 -13367.108} C_VEL
LIN {X 0,Y 401.256,Z 179.19,A -85,B 0,C 180,E1 -13368.998,E2 -13368.998} C_VEL
LIN {X 0,Y 402.906,Z 185.369,A -85,B 0,C 180,E1 -13370.321,E2 -13370.321} C_VEL
LIN {X 0,Y 401.89,Z 199.826,A -85,B 0,C 180,E1 -13371.25,E2 -13371.25} C_VEL
LIN {X 0,Y 391.637,Z 270.648,A -85,B 0,C 180,E1 -13373.607,E2 -13373.607} C_VEL
LIN {X 0,Y 384.344,Z 333.135,A -85,B 0,C 180,E1 -13375.658,E2 -13375.658} C_VEL
LIN {X 0,Y 381.748,Z 354.099,A -85,B 0,C 180,E1 -13376.421,E2 -13376.421} C_VEL
LIN {X 0,Y 378.523,Z 373.842,A -85,B 0,C 180,E1 -13377.343,E2 -13377.343} C_VEL
LIN {X 0,Y 375.802,Z 389.341,A -85,B 0,C 180,E1 -13378.265,E2 -13378.265} C_VEL
LIN {X 0,Y 372.5,Z 406.664,A -85,B 0,C 180,E1 -13379.531,E2 -13379.531} C_VEL
LIN {X 0,Y 369.258,Z 423.312,A -85,B 0,C 180,E1 -13381.027,E2 -13381.027} C_VEL
LIN {X 0,Y 366.275,Z 437.819,A -85,B 0,C 180,E1 -13382.58,E2 -13382.58} C_VEL
LIN {X 0,Y 363.464,Z 451.879,A -85,B 0,C 180,E1 -13384.364,E2 -13384.364} C_VEL
LIN {X 0,Y 361.12,Z 463.992,A -85,B 0,C 180,E1 -13386.162,E2 -13386.162} C_VEL
LIN {X 0,Y 358.943,Z 475.589,A -85,B 0,C 180,E1 -13388.159,E2 -13388.159} C_VEL
LIN {X 0,Y 356.998,Z 486.865,A -85,B 0,C 180,E1 -13390.447,E2 -13390.447} C_VEL
LIN {X 0,Y 355.582,Z 496.384,A -85,B 0,C 180,E1 -13392.753,E2 -13392.753} C_VEL
LIN {X 0,Y 354.518,Z 504.404,A -85,B 0,C 180,E1 -13395.065,E2 -13395.065} C_VEL
LIN {X 0,Y 353.902,Z 511.115,A -85,B 0,C 180,E1 -13397.382,E2 -13397.382} C_VEL
LIN {X 0,Y 353.461,Z 516.525,A -85,B 0,C 180,E1 -13399.691,E2 -13399.691} C_VEL
LIN {X 0,Y 353.439,Z 520.748,A -85,B 0,C 180,E1 -13401.998,E2 -13401.998} C_VEL
LIN {X 0,Y 353.485,Z 523.87,A -85,B 0,C 180,E1 -13404.294,E2 -13404.294} C_VEL
LIN {X 0,Y 353.5,Z 525.778,A -85,B 0,C 180,E1 -13406.58,E2 -13406.58} C_VEL
LIN {X 0,Y 353.624,Z 526.662,A -85,B 0,C 180,E1 -13408.86,E2 -13408.86} C_VEL
LIN {X 0,Y 353.716,Z 526.332,A -85,B 0,C 180,E1 -13411.138,E2 -13411.138} C_VEL
LIN {X 0,Y 353.609,Z 524.896,A -85,B 0,C 180,E1 -13413.418,E2 -13413.418} C_VEL
LIN {X 0,Y 353.622,Z 522.303,A -85,B 0,C 180,E1 -13415.702,E2 -13415.702} C_VEL
LIN {X 0,Y 353.532,Z 518.463,A -85,B 0,C 180,E1 -13417.998,E2 -13417.998} C_VEL
LIN {X 0,Y 353.541,Z 513.405,A -85,B 0,C 180,E1 -13420.305,E2 -13420.305} C_VEL
LIN {X 0,Y 353.916,Z 506.984,A -85,B 0,C 180,E1 -13422.616,E2 -13422.616} C_VEL
LIN {X 0,Y 354.357,Z 500.118,A -85,B 0,C 180,E1 -13424.647,E2 -13424.647} C_VEL
LIN {X 0,Y 355.068,Z 492.074,A -85,B 0,C 180,E1 -13426.678,E2 -13426.678} C_VEL
LIN {X 0,Y 356.005,Z 482.892,A -85,B 0,C 180,E1 -13428.634,E2 -13428.634} C_VEL
LIN {X 0,Y 357.373,Z 471.344,A -85,B 0,C 180,E1 -13430.73,E2 -13430.73} C_VEL
LIN {X 0,Y 358.923,Z 459.186,A -85,B 0,C 180,E1 -13432.598,E2 -13432.598} C_VEL
LIN {X 0,Y 360.573,Z 446.049,A -85,B 0,C 180,E1 -13434.314,E2 -13434.314} C_VEL
LIN {X 0,Y 362.397,Z 431.926,A -85,B 0,C 180,E1 -13435.87,E2 -13435.87} C_VEL
LIN {X 0,Y 364.216,Z 416.759,A -85,B 0,C 180,E1 -13437.264,E2 -13437.264} C_VEL
LIN {X 0,Y 366.147,Z 399.98,A -85,B 0,C 180,E1 -13438.519,E2 -13438.519} C_VEL
LIN {X 0,Y 367.872,Z 382.626,A -85,B 0,C 180,E1 -13439.546,E2 -13439.546} C_VEL
LIN {X 0,Y 369.434,Z 364.51,A -85,B 0,C 180,E1 -13440.351,E2 -13440.351} C_VEL
LIN {X 0,Y 370.535,Z 345.842,A -85,B 0,C 180,E1 -13440.933,E2 -13440.933} C_VEL
LIN {X 0,Y 377.506,Z 193.872,A -85,B 0,C 180,E1 -13444.768,E2 -13444.768} C_VEL
LIN {X 0,Y 373.815,Z 164.05,A -85,B 0,C 180,E1 -13445.949,E2 -13445.949} C_VEL
LIN {X 0,Y 365.822,Z 146.093,A -85,B 0,C 180,E1 -13447.188,E2 -13447.188} C_VEL
LIN {X 0,Y 358.866,Z 124.651,A -85,B 0,C 180,E1 -13450.665,E2 -13450.665} C_VEL
LIN {X 0,Y 354.834,Z 112.6,A -85,B 0,C 180,E1 -13452.762,E2 -13452.762} C_VEL
LIN {X 0,Y 354.779,Z 112.606,A -85,B 0,C 180,E1 -13456.106,E2 -13456.106} C_VEL
LIN {X 0,Y 354.784,Z 112.601,A -85,B 0,C 180,E1 -13459.179,E2 -13459.179} C_VEL
LIN {X 0,Y 354.808,Z 112.603,A -85,B 0,C 180,E1 -13462.401,E2 -13462.401} C_VEL
LIN {X 0,Y 354.808,Z 112.598,A -85,B 0,C 180,E1 -13464.941,E2 -13464.941} C_VEL
LIN {X 0,Y 354.81,Z 112.601,A -85,B 0,C 180,E1 -13468.399,E2 -13468.399} C_VEL
LIN {X 0,Y 354.849,Z 112.594,A -85,B 0,C 180,E1 -13471.619,E2 -13471.619} C_VEL
LIN {X 0,Y 354.895,Z 112.592,A -85,B 0,C 180,E1 -13474.172,E2 -13474.172} C_VEL
LIN {X 0,Y 354.83,Z 112.6,A -85,B 0,C 180,E1 -13477.894,E2 -13477.894} C_VEL
LIN {X 0,Y 354.918,Z 112.59,A -85,B 0,C 180,E1 -13481.891,E2 -13481.891} C_VEL
LIN {X 0,Y 354.939,Z 112.586,A -85,B 0,C 180,E1 -13485.98,E2 -13485.98} C_VEL
LIN {X 0,Y 354.978,Z 112.582,A -85,B 0,C 180,E1 -13489.736,E2 -13489.736} C_VEL
LIN {X 0,Y 355.109,Z 112.564,A -85,B 0,C 180,E1 -13492.037,E2 -13492.037} C_VEL
LIN {X 0,Y 355.088,Z 112.564,A -85,B 0,C 180,E1 -13494.321,E2 -13494.321} C_VEL
LIN {X 0,Y 355.241,Z 112.549,A -85,B 0,C 180,E1 -13497.732,E2 -13497.732} C_VEL
LIN {X 0,Y 355.393,Z 112.527,A -85,B 0,C 180,E1 -13500,E2 -13500} C_VEL
LIN {X 0,Y 355.241,Z 112.544,A -85,B 0,C 180,E1 -13502.268,E2 -13502.268} C_VEL
LIN {X 0,Y 355.133,Z 112.558,A -85,B 0,C 180,E1 -13506.819,E2 -13506.819} C_VEL
LIN {X 0,Y 355.011,Z 112.575,A -85,B 0,C 180,E1 -13509.113,E2 -13509.113} C_VEL
LIN {X 0,Y 354.917,Z 112.584,A -85,B 0,C 180,E1 -13512.581,E2 -13512.581} C_VEL
LIN {X 0,Y 354.885,Z 112.588,A -85,B 0,C 180,E1 -13516.096,E2 -13516.096} C_VEL
LIN {X 0,Y 354.897,Z 112.587,A -85,B 0,C 180,E1 -13518.472,E2 -13518.472} C_VEL
LIN {X 0,Y 354.83,Z 112.595,A -85,B 0,C 180,E1 -13522.106,E2 -13522.106} C_VEL
LIN {X 0,Y 354.895,Z 112.588,A -85,B 0,C 180,E1 -13525.828,E2 -13525.828} C_VEL
LIN {X 0,Y 354.813,Z 112.598,A -85,B 0,C 180,E1 -13529.682,E2 -13529.682} C_VEL
LIN {X 0,Y 354.802,Z 112.599,A -85,B 0,C 180,E1 -13533.702,E2 -13533.702} C_VEL
LIN {X 0,Y 354.795,Z 112.601,A -85,B 0,C 180,E1 -13536.46,E2 -13536.46} C_VEL
LIN {X 0,Y 354.82,Z 112.598,A -85,B 0,C 180,E1 -13539.424,E2 -13539.424} C_VEL
LIN {X 0,Y 354.785,Z 112.607,A -85,B 0,C 180,E1 -13542.868,E2 -13542.868} C_VEL
LIN {X 0,Y 354.782,Z 112.601,A -85,B 0,C 180,E1 -13546.107,E2 -13546.107} C_VEL
LIN {X 0,Y 354.822,Z 112.598,A -85,B 0,C 180,E1 -13549.185,E2 -13549.185} C_VEL
LIN {X 0,Y 354.809,Z 112.601,A -85,B 0,C 180,E1 -13552.402,E2 -13552.402} C_VEL
LIN {X 0,Y 354.809,Z 112.601,A -85,B 0,C 180,E1 -13554.942,E2 -13554.942} C_VEL
LIN {X 0,Y 354.791,Z 112.604,A -85,B 0,C 180,E1 -13558.406,E2 -13558.406} C_VEL
LIN {X 0,Y 354.844,Z 112.593,A -85,B 0,C 180,E1 -13561.619,E2 -13561.619} C_VEL
LIN {X 0,Y 354.898,Z 112.589,A -85,B 0,C 180,E1 -13564.173,E2 -13564.173} C_VEL
LIN {X 0,Y 354.838,Z 112.595,A -85,B 0,C 180,E1 -13567.895,E2 -13567.895} C_VEL
LIN {X 0,Y 354.923,Z 112.585,A -85,B 0,C 180,E1 -13571.892,E2 -13571.892} C_VEL
LIN {X 0,Y 354.942,Z 112.584,A -85,B 0,C 180,E1 -13575.982,E2 -13575.982} C_VEL
LIN {X 0,Y 354.979,Z 112.578,A -85,B 0,C 180,E1 -13579.737,E2 -13579.737} C_VEL
LIN {X 0,Y 355.115,Z 112.564,A -85,B 0,C 180,E1 -13582.038,E2 -13582.038} C_VEL
LIN {X 0,Y 355.092,Z 112.567,A -85,B 0,C 180,E1 -13584.321,E2 -13584.321} C_VEL
LIN {X 0,Y 355.244,Z 112.546,A -85,B 0,C 180,E1 -13587.733,E2 -13587.733} C_VEL
LIN {X 0,Y 355.397,Z 112.53,A -85,B 0,C 180,E1 -13590.001,E2 -13590.001} C_VEL
LIN {X 0,Y 355.244,Z 112.547,A -85,B 0,C 180,E1 -13592.268,E2 -13592.268} C_VEL
LIN {X 0,Y 355.139,Z 112.556,A -85,B 0,C 180,E1 -13596.82,E2 -13596.82} C_VEL
LIN {X 0,Y 355.017,Z 112.572,A -85,B 0,C 180,E1 -13599.113,E2 -13599.113} C_VEL
LIN {X 0,Y 354.923,Z 112.584,A -85,B 0,C 180,E1 -13602.582,E2 -13602.582} C_VEL
LIN {X 0,Y 354.891,Z 112.59,A -85,B 0,C 180,E1 -13606.097,E2 -13606.097} C_VEL
LIN {X 0,Y 354.903,Z 112.586,A -85,B 0,C 180,E1 -13608.473,E2 -13608.473} C_VEL
LIN {X 0,Y 354.837,Z 112.596,A -85,B 0,C 180,E1 -13612.107,E2 -13612.107} C_VEL
LIN {X 0,Y 354.901,Z 112.59,A -85,B 0,C 180,E1 -13615.828,E2 -13615.828} C_VEL
LIN {X 0,Y 354.82,Z 112.601,A -85,B 0,C 180,E1 -13619.682,E2 -13619.682} C_VEL
LIN {X 0,Y 354.809,Z 112.601,A -85,B 0,C 180,E1 -13623.703,E2 -13623.703} C_VEL
LIN {X 0,Y 354.803,Z 112.598,A -85,B 0,C 180,E1 -13626.46,E2 -13626.46} C_VEL
LIN {X 0,Y 354.827,Z 112.601,A -85,B 0,C 180,E1 -13629.424,E2 -13629.424} C_VEL
LIN {X 0,Y 354.792,Z 112.602,A -85,B 0,C 180,E1 -13632.868,E2 -13632.868} C_VEL
LIN {X 0,Y 354.784,Z 112.601,A -85,B 0,C 180,E1 -13636.106,E2 -13636.106} C_VEL
LIN {X 0,Y 354.78,Z 112.603,A -85,B 0,C 180,E1 -13639.599,E2 -13639.599} C_VEL
LIN {X 0,Y 354.786,Z 112.598,A -85,B 0,C 180,E1 -13641.324,E2 -13641.324} C_VEL
LIN {X 0,Y 354.856,Z 113.352,A -85,B 0,C 180,E1 -13641.825,E2 -13641.825} C_VEL
LIN {X 0,Y 355.118,Z 115.804,A -85,B 0,C 180,E1 -13642.37,E2 -13642.37} C_VEL
LIN {X 0,Y 355.712,Z 120.55,A -85,B 0,C 180,E1 -13642.923,E2 -13642.923} C_VEL
LIN {X 0,Y 356.716,Z 126.428,A -85,B 0,C 180,E1 -13643.311,E2 -13643.311} C_VEL
LIN {X 0,Y 359.427,Z 136.647,A -85,B 0,C 180,E1 -13643.876,E2 -13643.876} C_VEL
LIN {X 0,Y 360.243,Z 138.546,A -85,B 0,C 180,E1 -13644.007,E2 -13644.007} C_VEL
LIN {X 0,Y 370.514,Z 159.321,A -85,B 0,C 180,E1 -13645.5,E2 -13645.5} C_VEL
LIN {X 0,Y 364.266,Z 291.083,A -85,B 0,C 180,E1 -13648.888,E2 -13648.888} C_VEL
LIN {X 0,Y 363.328,Z 309.811,A -85,B 0,C 180,E1 -13649.485,E2 -13649.485} C_VEL
LIN {X 0,Y 362.135,Z 328.359,A -85,B 0,C 180,E1 -13650.338,E2 -13650.338} C_VEL
LIN {X 0,Y 360.738,Z 344.492,A -85,B 0,C 180,E1 -13651.306,E2 -13651.306} C_VEL
LIN {X 0,Y 359.281,Z 360.111,A -85,B 0,C 180,E1 -13652.475,E2 -13652.475} C_VEL
LIN {X 0,Y 357.709,Z 374.455,A -85,B 0,C 180,E1 -13653.764,E2 -13653.764} C_VEL
LIN {X 0,Y 355.961,Z 388.524,A -85,B 0,C 180,E1 -13655.261,E2 -13655.261} C_VEL
LIN {X 0,Y 354.283,Z 401.817,A -85,B 0,C 180,E1 -13656.934,E2 -13656.934} C_VEL
LIN {X 0,Y 352.721,Z 413.592,A -85,B 0,C 180,E1 -13658.676,E2 -13658.676} C_VEL
LIN {X 0,Y 351.46,Z 423.763,A -85,B 0,C 180,E1 -13660.431,E2 -13660.431} C_VEL
LIN {X 0,Y 350.137,Z 434.026,A -85,B 0,C 180,E1 -13662.477,E2 -13662.477} C_VEL
LIN {X 0,Y 348.968,Z 443.92,A -85,B 0,C 180,E1 -13664.822,E2 -13664.822} C_VEL
LIN {X 0,Y 348.06,Z 452.14,A -85,B 0,C 180,E1 -13667.167,E2 -13667.167} C_VEL
LIN {X 0,Y 347.404,Z 458.852,A -85,B 0,C 180,E1 -13669.51,E2 -13669.51} C_VEL
LIN {X 0,Y 347.021,Z 464.29,A -85,B 0,C 180,E1 -13671.85,E2 -13671.85} C_VEL
LIN {X 0,Y 346.754,Z 468.567,A -85,B 0,C 180,E1 -13674.184,E2 -13674.184} C_VEL
LIN {X 0,Y 346.677,Z 471.621,A -85,B 0,C 180,E1 -13676.513,E2 -13676.513} C_VEL
LIN {X 0,Y 346.555,Z 473.679,A -85,B 0,C 180,E1 -13678.838,E2 -13678.838} C_VEL
LIN {X 0,Y 346.679,Z 474.673,A -85,B 0,C 180,E1 -13681.161,E2 -13681.161} C_VEL
LIN {X 0,Y 346.949,Z 474.612,A -85,B 0,C 180,E1 -13683.484,E2 -13683.484} C_VEL
LIN {X 0,Y 347.209,Z 473.594,A -85,B 0,C 180,E1 -13685.809,E2 -13685.809} C_VEL
LIN {X 0,Y 347.695,Z 471.46,A -85,B 0,C 180,E1 -13688.134,E2 -13688.134} C_VEL
LIN {X 0,Y 348.473,Z 468.333,A -85,B 0,C 180,E1 -13690.458,E2 -13690.458} C_VEL
LIN {X 0,Y 349.487,Z 464.068,A -85,B 0,C 180,E1 -13692.78,E2 -13692.78} C_VEL
LIN {X 0,Y 350.67,Z 458.676,A -85,B 0,C 180,E1 -13695.102,E2 -13695.102} C_VEL
LIN {X 0,Y 352.412,Z 452.033,A -85,B 0,C 180,E1 -13697.406,E2 -13697.406} C_VEL
LIN {X 0,Y 354.47,Z 444,A -85,B 0,C 180,E1 -13699.697,E2 -13699.697} C_VEL
LIN {X 0,Y 356.959,Z 434.35,A -85,B 0,C 180,E1 -13701.967,E2 -13701.967} C_VEL
LIN {X 0,Y 359.823,Z 422.907,A -85,B 0,C 180,E1 -13704.215,E2 -13704.215} C_VEL
LIN {X 0,Y 362.722,Z 411.085,A -85,B 0,C 180,E1 -13706.155,E2 -13706.155} C_VEL
LIN {X 0,Y 366.068,Z 397.186,A -85,B 0,C 180,E1 -13708.057,E2 -13708.057} C_VEL
LIN {X 0,Y 368.572,Z 385.68,A -85,B 0,C 180,E1 -13709.406,E2 -13709.406} C_VEL
LIN {X 0,Y 371.606,Z 371.122,A -85,B 0,C 180,E1 -13710.853,E2 -13710.853} C_VEL
LIN {X 0,Y 374.634,Z 355.188,A -85,B 0,C 180,E1 -13712.164,E2 -13712.164} C_VEL
LIN {X 0,Y 377.497,Z 338.013,A -85,B 0,C 180,E1 -13713.313,E2 -13713.313} C_VEL
LIN {X 0,Y 379.916,Z 321.46,A -85,B 0,C 180,E1 -13714.187,E2 -13714.187} C_VEL
LIN {X 0,Y 381.831,Z 305.966,A -85,B 0,C 180,E1 -13714.831,E2 -13714.831} C_VEL
LIN {X 0,Y 390.161,Z 246.641,A -85,B 0,C 180,E1 -13716.874,E2 -13716.874} C_VEL
LIN {X 0,Y 401.329,Z 180.882,A -85,B 0,C 180,E1 -13719.142,E2 -13719.142} C_VEL
LIN {X 0,Y 399.947,Z 178.352,A -85,B 0,C 180,E1 -13720.132,E2 -13720.132} C_VEL
LIN {X 0,Y 398.079,Z 175.856,A -85,B 0,C 180,E1 -13721.913,E2 -13721.913} C_VEL
LIN {X 0,Y 397.03,Z 175.692,A -85,B 0,C 180,E1 -13723.815,E2 -13723.815} C_VEL
LIN {X 0,Y 397.005,Z 177.572,A -85,B 0,C 180,E1 -13725.673,E2 -13725.673} C_VEL
LIN {X 0,Y 397.558,Z 180.122,A -85,B 0,C 180,E1 -13726.962,E2 -13726.962} C_VEL
LIN {X 0,Y 398.89,Z 185.655,A -85,B 0,C 180,E1 -13728.684,E2 -13728.684} C_VEL
LIN {X 0,Y 399.864,Z 189.902,A -85,B 0,C 180,E1 -13729.617,E2 -13729.617} C_VEL
LIN {X 0,Y 398.674,Z 201.932,A -85,B 0,C 180,E1 -13730.381,E2 -13730.381} C_VEL
LIN {X 0,Y 387.574,Z 273.056,A -85,B 0,C 180,E1 -13732.797,E2 -13732.797} C_VEL
LIN {X 0,Y 378.036,Z 347.299,A -85,B 0,C 180,E1 -13735.335,E2 -13735.335} C_VEL
LIN {X 0,Y 374.899,Z 366.494,A -85,B 0,C 180,E1 -13736.183,E2 -13736.183} C_VEL
LIN {X 0,Y 371.398,Z 384.71,A -85,B 0,C 180,E1 -13737.202,E2 -13737.202} C_VEL
LIN {X 0,Y 367.938,Z 402.327,A -85,B 0,C 180,E1 -13738.473,E2 -13738.473} C_VEL
LIN {X 0,Y 364.435,Z 418.782,A -85,B 0,C 180,E1 -13739.907,E2 -13739.907} C_VEL
LIN {X 0,Y 360.97,Z 434.611,A -85,B 0,C 180,E1 -13741.568,E2 -13741.568} C_VEL
LIN {X 0,Y 357.722,Z 449.56,A -85,B 0,C 180,E1 -13743.451,E2 -13743.451} C_VEL
LIN {X 0,Y 354.922,Z 462.805,A -85,B 0,C 180,E1 -13745.428,E2 -13745.428} C_VEL
LIN {X 0,Y 352.62,Z 474.319,A -85,B 0,C 180,E1 -13747.438,E2 -13747.438} C_VEL
LIN {X 0,Y 350.44,Z 485.619,A -85,B 0,C 180,E1 -13749.76,E2 -13749.76} C_VEL
LIN {X 0,Y 348.834,Z 495.193,A -85,B 0,C 180,E1 -13752.106,E2 -13752.106} C_VEL
LIN {X 0,Y 347.799,Z 502.375,A -85,B 0,C 180,E1 -13754.169,E2 -13754.169} C_VEL
LIN {X 0,Y 347.066,Z 508.958,A -85,B 0,C 180,E1 -13756.405,E2 -13756.405} C_VEL
LIN {X 0,Y 346.517,Z 514.929,A -85,B 0,C 180,E1 -13758.89,E2 -13758.89} C_VEL
LIN {X 0,Y 346.333,Z 518.392,A -85,B 0,C 180,E1 -13760.656,E2 -13760.656} C_VEL
LIN {X 0,Y 346.396,Z 521.994,A -85,B 0,C 180,E1 -13763.007,E2 -13763.007} C_VEL
LIN {X 0,Y 346.393,Z 524.461,A -85,B 0,C 180,E1 -13765.344,E2 -13765.344} C_VEL
LIN {X 0,Y 346.555,Z 525.786,A -85,B 0,C 180,E1 -13767.675,E2 -13767.675} C_VEL
LIN {X 0,Y 346.639,Z 526.042,A -85,B 0,C 180,E1 -13769.999,E2 -13769.999} C_VEL
LIN {X 0,Y 346.583,Z 525.058,A -85,B 0,C 180,E1 -13772.324,E2 -13772.324} C_VEL
LIN {X 0,Y 346.43,Z 522.987,A -85,B 0,C 180,E1 -13774.654,E2 -13774.654} C_VEL
LIN {X 0,Y 346.537,Z 520.622,A -85,B 0,C 180,E1 -13776.411,E2 -13776.411} C_VEL
LIN {X 0,Y 346.431,Z 516.451,A -85,B 0,C 180,E1 -13778.751,E2 -13778.751} C_VEL
LIN {X 0,Y 346.569,Z 510.896,A -85,B 0,C 180,E1 -13781.107,E2 -13781.107} C_VEL
LIN {X 0,Y 347.027,Z 503.666,A -85,B 0,C 180,E1 -13783.568,E2 -13783.568} C_VEL
LIN {X 0,Y 347.65,Z 495.553,A -85,B 0,C 180,E1 -13785.837,E2 -13785.837} C_VEL
LIN {X 0,Y 348.556,Z 486.77,A -85,B 0,C 180,E1 -13787.907,E2 -13787.907} C_VEL
LIN {X 0,Y 349.698,Z 476.368,A -85,B 0,C 180,E1 -13789.977,E2 -13789.977} C_VEL
LIN {X 0,Y 351.254,Z 464.182,A -85,B 0,C 180,E1 -13792.033,E2 -13792.033} C_VEL
LIN {X 0,Y 352.972,Z 451.181,A -85,B 0,C 180,E1 -13793.886,E2 -13793.886} C_VEL
LIN {X 0,Y 354.707,Z 437.598,A -85,B 0,C 180,E1 -13795.527,E2 -13795.527} C_VEL
LIN {X 0,Y 356.536,Z 423.523,A -85,B 0,C 180,E1 -13796.959,E2 -13796.959} C_VEL
LIN {X 0,Y 358.409,Z 408.455,A -85,B 0,C 180,E1 -13798.232,E2 -13798.232} C_VEL
LIN {X 0,Y 360.17,Z 392.128,A -85,B 0,C 180,E1 -13799.357,E2 -13799.357} C_VEL
LIN {X 0,Y 361.822,Z 375.548,A -85,B 0,C 180,E1 -13800.251,E2 -13800.251} C_VEL
LIN {X 0,Y 363.199,Z 358.863,A -85,B 0,C 180,E1 -13800.929,E2 -13800.929} C_VEL
LIN {X 0,Y 364.344,Z 336.257,A -85,B 0,C 180,E1 -13801.576,E2 -13801.576} C_VEL
LIN {X 0,Y 371.171,Z 194.603,A -85,B 0,C 180,E1 -13805.249,E2 -13805.249} C_VEL
LIN {X 0,Y 367.793,Z 166.737,A -85,B 0,C 180,E1 -13806.371,E2 -13806.371} C_VEL
LIN {X 0,Y 358.222,Z 145.442,A -85,B 0,C 180,E1 -13807.901,E2 -13807.901} C_VEL
LIN {X 0,Y 352.145,Z 126.456,A -85,B 0,C 180,E1 -13811.042,E2 -13811.042} C_VEL
LIN {X 0,Y 347.781,Z 113.476,A -85,B 0,C 180,E1 -13813.366,E2 -13813.366} C_VEL
LIN {X 0,Y 347.725,Z 113.483,A -85,B 0,C 180,E1 -13816.685,E2 -13816.685} C_VEL
LIN {X 0,Y 347.743,Z 113.482,A -85,B 0,C 180,E1 -13820.173,E2 -13820.173} C_VEL
LIN {X 0,Y 347.761,Z 113.478,A -85,B 0,C 180,E1 -13822.679,E2 -13822.679} C_VEL
LIN {X 0,Y 347.743,Z 113.481,A -85,B 0,C 180,E1 -13825.956,E2 -13825.956} C_VEL
LIN {X 0,Y 347.766,Z 113.476,A -85,B 0,C 180,E1 -13829.654,E2 -13829.654} C_VEL
LIN {X 0,Y 347.848,Z 113.465,A -85,B 0,C 180,E1 -13832.744,E2 -13832.744} C_VEL
LIN {X 0,Y 347.784,Z 113.478,A -85,B 0,C 180,E1 -13836.162,E2 -13836.162} C_VEL
LIN {X 0,Y 347.813,Z 113.475,A -85,B 0,C 180,E1 -13839.91,E2 -13839.91} C_VEL
LIN {X 0,Y 347.863,Z 113.465,A -85,B 0,C 180,E1 -13842.359,E2 -13842.359} C_VEL
LIN {X 0,Y 347.893,Z 113.464,A -85,B 0,C 180,E1 -13845.971,E2 -13845.971} C_VEL
LIN {X 0,Y 347.928,Z 113.458,A -85,B 0,C 180,E1 -13849.526,E2 -13849.526} C_VEL
LIN {X 0,Y 348.07,Z 113.442,A -85,B 0,C 180,E1 -13851.875,E2 -13851.875} C_VEL
LIN {X 0,Y 348.063,Z 113.44,A -85,B 0,C 180,E1 -13854.206,E2 -13854.206} C_VEL
LIN {X 0,Y 348.204,Z 113.426,A -85,B 0,C 180,E1 -13857.687,E2 -13857.687} C_VEL
LIN {X 0,Y 348.363,Z 113.403,A -85,B 0,C 180,E1 -13860,E2 -13860} C_VEL
LIN {X 0,Y 348.204,Z 113.421,A -85,B 0,C 180,E1 -13862.314,E2 -13862.314} C_VEL
LIN {X 0,Y 348.103,Z 113.434,A -85,B 0,C 180,E1 -13866.958,E2 -13866.958} C_VEL
LIN {X 0,Y 347.924,Z 113.455,A -85,B 0,C 180,E1 -13870.475,E2 -13870.475} C_VEL
LIN {X 0,Y 347.894,Z 113.459,A -85,B 0,C 180,E1 -13874.15,E2 -13874.15} C_VEL
LIN {X 0,Y 347.886,Z 113.46,A -85,B 0,C 180,E1 -13878.29,E2 -13878.29} C_VEL
LIN {X 0,Y 347.784,Z 113.475,A -85,B 0,C 180,E1 -13881.635,E2 -13881.635} C_VEL
LIN {X 0,Y 347.809,Z 113.475,A -85,B 0,C 180,E1 -13885.109,E2 -13885.109} C_VEL
LIN {X 0,Y 347.804,Z 113.471,A -85,B 0,C 180,E1 -13887.694,E2 -13887.694} C_VEL
LIN {X 0,Y 347.745,Z 113.478,A -85,B 0,C 180,E1 -13890.348,E2 -13890.348} C_VEL
LIN {X 0,Y 347.744,Z 113.478,A -85,B 0,C 180,E1 -13894.044,E2 -13894.044} C_VEL
LIN {X 0,Y 347.759,Z 113.478,A -85,B 0,C 180,E1 -13897.321,E2 -13897.321} C_VEL
LIN {X 0,Y 347.729,Z 113.48,A -85,B 0,C 180,E1 -13900.298,E2 -13900.298} C_VEL
LIN {X 0,Y 347.722,Z 113.482,A -85,B 0,C 180,E1 -13903.408,E2 -13903.408} C_VEL
LIN {X 0,Y 347.762,Z 113.48,A -85,B 0,C 180,E1 -13906.68,E2 -13906.68} C_VEL
LIN {X 0,Y 347.755,Z 113.477,A -85,B 0,C 180,E1 -13910.172,E2 -13910.172} C_VEL
LIN {X 0,Y 347.763,Z 113.481,A -85,B 0,C 180,E1 -13912.68,E2 -13912.68} C_VEL
LIN {X 0,Y 347.745,Z 113.478,A -85,B 0,C 180,E1 -13915.957,E2 -13915.957} C_VEL
LIN {X 0,Y 347.747,Z 113.477,A -85,B 0,C 180,E1 -13919.653,E2 -13919.653} C_VEL
LIN {X 0,Y 347.829,Z 113.467,A -85,B 0,C 180,E1 -13923.608,E2 -13923.608} C_VEL
LIN {X 0,Y 347.788,Z 113.475,A -85,B 0,C 180,E1 -13926.163,E2 -13926.163} C_VEL
LIN {X 0,Y 347.827,Z 113.469,A -85,B 0,C 180,E1 -13929.911,E2 -13929.911} C_VEL
LIN {X 0,Y 347.866,Z 113.469,A -85,B 0,C 180,E1 -13932.36,E2 -13932.36} C_VEL
LIN {X 0,Y 347.897,Z 113.461,A -85,B 0,C 180,E1 -13935.972,E2 -13935.972} C_VEL
LIN {X 0,Y 347.93,Z 113.455,A -85,B 0,C 180,E1 -13939.526,E2 -13939.526} C_VEL
LIN {X 0,Y 348.075,Z 113.439,A -85,B 0,C 180,E1 -13941.876,E2 -13941.876} C_VEL
LIN {X 0,Y 348.068,Z 113.443,A -85,B 0,C 180,E1 -13944.206,E2 -13944.206} C_VEL
LIN {X 0,Y 348.207,Z 113.422,A -85,B 0,C 180,E1 -13947.687,E2 -13947.687} C_VEL
LIN {X 0,Y 348.345,Z 113.408,A -85,B 0,C 180,E1 -13950.001,E2 -13950.001} C_VEL
LIN {X 0,Y 348.207,Z 113.423,A -85,B 0,C 180,E1 -13952.314,E2 -13952.314} C_VEL
LIN {X 0,Y 348.108,Z 113.432,A -85,B 0,C 180,E1 -13956.958,E2 -13956.958} C_VEL
LIN {X 0,Y 347.969,Z 113.451,A -85,B 0,C 180,E1 -13959.299,E2 -13959.299} C_VEL
LIN {X 0,Y 347.892,Z 113.459,A -85,B 0,C 180,E1 -13962.84,E2 -13962.84} C_VEL
LIN {X 0,Y 347.841,Z 113.466,A -85,B 0,C 180,E1 -13966.432,E2 -13966.432} C_VEL
LIN {X 0,Y 347.853,Z 113.464,A -85,B 0,C 180,E1 -13968.861,E2 -13968.861} C_VEL
LIN {X 0,Y 347.776,Z 113.474,A -85,B 0,C 180,E1 -13972.58,E2 -13972.58} C_VEL
LIN {X 0,Y 347.814,Z 113.47,A -85,B 0,C 180,E1 -13975.109,E2 -13975.109} C_VEL
LIN {X 0,Y 347.81,Z 113.474,A -85,B 0,C 180,E1 -13977.695,E2 -13977.695} C_VEL
LIN {X 0,Y 347.751,Z 113.477,A -85,B 0,C 180,E1 -13980.348,E2 -13980.348} C_VEL
LIN {X 0,Y 347.751,Z 113.478,A -85,B 0,C 180,E1 -13984.044,E2 -13984.044} C_VEL
LIN {X 0,Y 347.768,Z 113.48,A -85,B 0,C 180,E1 -13987.321,E2 -13987.321} C_VEL
LIN {X 0,Y 347.735,Z 113.479,A -85,B 0,C 180,E1 -13990.297,E2 -13990.297} C_VEL
LIN {X 0,Y 347.727,Z 113.485,A -85,B 0,C 180,E1 -13993.408,E2 -13993.408} C_VEL
LIN {X 0,Y 347.731,Z 113.48,A -85,B 0,C 180,E1 -13996.686,E2 -13996.686} C_VEL
LIN {X 0,Y 347.75,Z 113.477,A -85,B 0,C 180,E1 -14000.173,E2 -14000.173} C_VEL
LIN {X 0,Y 347.762,Z 113.475,A -85,B 0,C 180,E1 -14002.051,E2 -14002.051} C_VEL
LIN {X 0,Y 348.905,Z 116.541,A -85,B 0,C 180,E1 -14002.275,E2 -14002.275} C_VEL
LIN {X 0,Y 360.243,Z 138.546,A -85,B 0,C 180,E1 -14004.007,E2 -14004.007} C_VEL
LIN {X 0,Y 362.173,Z 143.757,A -85,B 0,C 180,E1 -14004.336,E2 -14004.336} C_VEL
LIN {X 0,Y 363.324,Z 149.337,A -85,B 0,C 180,E1 -14004.607,E2 -14004.607} C_VEL
LIN {X 0,Y 363.743,Z 153.166,A -85,B 0,C 180,E1 -14004.76,E2 -14004.76} C_VEL
LIN {X 0,Y 363.995,Z 161.048,A -85,B 0,C 180,E1 -14005.024,E2 -14005.024} C_VEL
LIN {X 0,Y 363.812,Z 168.986,A -85,B 0,C 180,E1 -14005.252,E2 -14005.252} C_VEL
LIN {X 0,Y 357.24,Z 301.821,A -85,B 0,C 180,E1 -14008.784,E2 -14008.784} C_VEL
LIN {X 0,Y 356.206,Z 318.976,A -85,B 0,C 180,E1 -14009.466,E2 -14009.466} C_VEL
LIN {X 0,Y 354.82,Z 336.783,A -85,B 0,C 180,E1 -14010.418,E2 -14010.418} C_VEL
LIN {X 0,Y 353.381,Z 352.465,A -85,B 0,C 180,E1 -14011.49,E2 -14011.49} C_VEL
LIN {X 0,Y 351.686,Z 368.153,A -85,B 0,C 180,E1 -14012.798,E2 -14012.798} C_VEL
LIN {X 0,Y 349.817,Z 383.099,A -85,B 0,C 180,E1 -14014.297,E2 -14014.297} C_VEL
LIN {X 0,Y 348.029,Z 397.422,A -85,B 0,C 180,E1 -14016.021,E2 -14016.021} C_VEL
LIN {X 0,Y 346.218,Z 410.871,A -85,B 0,C 180,E1 -14017.942,E2 -14017.942} C_VEL
LIN {X 0,Y 344.626,Z 423.157,A -85,B 0,C 180,E1 -14020.026,E2 -14020.026} C_VEL
LIN {X 0,Y 343.238,Z 433.623,A -85,B 0,C 180,E1 -14022.113,E2 -14022.113} C_VEL
LIN {X 0,Y 342.024,Z 443.685,A -85,B 0,C 180,E1 -14024.507,E2 -14024.507} C_VEL
LIN {X 0,Y 341.08,Z 452.016,A -85,B 0,C 180,E1 -14026.9,E2 -14026.9} C_VEL
LIN {X 0,Y 340.373,Z 458.88,A -85,B 0,C 180,E1 -14029.29,E2 -14029.29} C_VEL
LIN {X 0,Y 339.982,Z 464.462,A -85,B 0,C 180,E1 -14031.68,E2 -14031.68} C_VEL
LIN {X 0,Y 339.689,Z 468.828,A -85,B 0,C 180,E1 -14034.062,E2 -14034.062} C_VEL
LIN {X 0,Y 339.587,Z 472.005,A -85,B 0,C 180,E1 -14036.44,E2 -14036.44} C_VEL
LIN {X 0,Y 339.49,Z 474.18,A -85,B 0,C 180,E1 -14038.814,E2 -14038.814} C_VEL
LIN {X 0,Y 339.609,Z 475.241,A -85,B 0,C 180,E1 -14041.186,E2 -14041.186} C_VEL
LIN {X 0,Y 339.896,Z 475.299,A -85,B 0,C 180,E1 -14043.556,E2 -14043.556} C_VEL
LIN {X 0,Y 340.175,Z 474.351,A -85,B 0,C 180,E1 -14045.929,E2 -14045.929} C_VEL
LIN {X 0,Y 340.726,Z 472.337,A -85,B 0,C 180,E1 -14048.302,E2 -14048.302} C_VEL
LIN {X 0,Y 341.551,Z 469.333,A -85,B 0,C 180,E1 -14050.672,E2 -14050.672} C_VEL
LIN {X 0,Y 342.919,Z 463.998,A -85,B 0,C 180,E1 -14053.632,E2 -14053.632} C_VEL
LIN {X 0,Y 344.391,Z 458.394,A -85,B 0,C 180,E1 -14055.991,E2 -14055.991} C_VEL
LIN {X 0,Y 346.264,Z 451.551,A -85,B 0,C 180,E1 -14058.336,E2 -14058.336} C_VEL
LIN {X 0,Y 348.546,Z 443.329,A -85,B 0,C 180,E1 -14060.662,E2 -14060.662} C_VEL
LIN {X 0,Y 351.372,Z 433.403,A -85,B 0,C 180,E1 -14062.98,E2 -14062.98} C_VEL
LIN {X 0,Y 354.5,Z 421.861,A -85,B 0,C 180,E1 -14065.229,E2 -14065.229} C_VEL
LIN {X 0,Y 357.618,Z 410.202,A -85,B 0,C 180,E1 -14067.131,E2 -14067.131} C_VEL
LIN {X 0,Y 361.283,Z 395.723,A -85,B 0,C 180,E1 -14069.099,E2 -14069.099} C_VEL
LIN {X 0,Y 364.343,Z 382.787,A -85,B 0,C 180,E1 -14070.581,E2 -14070.581} C_VEL
LIN {X 0,Y 367.348,Z 369.145,A -85,B 0,C 180,E1 -14071.905,E2 -14071.905} C_VEL
LIN {X 0,Y 370.512,Z 353.603,A -85,B 0,C 180,E1 -14073.164,E2 -14073.164} C_VEL
LIN {X 0,Y 373.472,Z 336.822,A -85,B 0,C 180,E1 -14074.288,E2 -14074.288} C_VEL
LIN {X 0,Y 376.278,Z 318.897,A -85,B 0,C 180,E1 -14075.217,E2 -14075.217} C_VEL
LIN {X 0,Y 379.874,Z 292.668,A -85,B 0,C 180,E1 -14076.219,E2 -14076.219} C_VEL
LIN {X 0,Y 390.203,Z 229.044,A -85,B 0,C 180,E1 -14078.458,E2 -14078.458} C_VEL
LIN {X 0,Y 398.302,Z 185.806,A -85,B 0,C 180,E1 -14079.965,E2 -14079.965} C_VEL
LIN {X 0,Y 396.844,Z 183.653,A -85,B 0,C 180,E1 -14081.227,E2 -14081.227} C_VEL
LIN {X 0,Y 396.05,Z 182.512,A -85,B 0,C 180,E1 -14082.237,E2 -14082.237} C_VEL
LIN {X 0,Y 395.248,Z 182.573,A -85,B 0,C 180,E1 -14083.767,E2 -14083.767} C_VEL
LIN {X 0,Y 395.159,Z 184.443,A -85,B 0,C 180,E1 -14085.596,E2 -14085.596} C_VEL
LIN {X 0,Y 395.5,Z 186.553,A -85,B 0,C 180,E1 -14086.643,E2 -14086.643} C_VEL
LIN {X 0,Y 396.513,Z 191.651,A -85,B 0,C 180,E1 -14088.266,E2 -14088.266} C_VEL
LIN {X 0,Y 396.981,Z 194.392,A -85,B 0,C 180,E1 -14088.871,E2 -14088.871} C_VEL
LIN {X 0,Y 395.862,Z 203.703,A -85,B 0,C 180,E1 -14089.47,E2 -14089.47} C_VEL
LIN {X 0,Y 383.904,Z 274.595,A -85,B 0,C 180,E1 -14091.923,E2 -14091.923} C_VEL
LIN {X 0,Y 373.813,Z 346.214,A -85,B 0,C 180,E1 -14094.432,E2 -14094.432} C_VEL
LIN {X 0,Y 370.418,Z 365.554,A -85,B 0,C 180,E1 -14095.305,E2 -14095.305} C_VEL
LIN {X 0,Y 366.942,Z 382.472,A -85,B 0,C 180,E1 -14096.259,E2 -14096.259} C_VEL
LIN {X 0,Y 363.175,Z 400.078,A -85,B 0,C 180,E1 -14097.519,E2 -14097.519} C_VEL
LIN {X 0,Y 359.424,Z 416.525,A -85,B 0,C 180,E1 -14098.953,E2 -14098.953} C_VEL
LIN {X 0,Y 355.926,Z 431.463,A -85,B 0,C 180,E1 -14100.515,E2 -14100.515} C_VEL
LIN {X 0,Y 352.912,Z 444.339,A -85,B 0,C 180,E1 -14102.096,E2 -14102.096} C_VEL
LIN {X 0,Y 349.7,Z 458.073,A -85,B 0,C 180,E1 -14104.079,E2 -14104.079} C_VEL
LIN {X 0,Y 346.963,Z 469.986,A -85,B 0,C 180,E1 -14106.101,E2 -14106.101} C_VEL
LIN {X 0,Y 344.499,Z 481.751,A -85,B 0,C 180,E1 -14108.455,E2 -14108.455} C_VEL
LIN {X 0,Y 342.533,Z 491.815,A -85,B 0,C 180,E1 -14110.835,E2 -14110.835} C_VEL
LIN {X 0,Y 341.144,Z 500.368,A -85,B 0,C 180,E1 -14113.236,E2 -14113.236} C_VEL
LIN {X 0,Y 340.03,Z 509.148,A -85,B 0,C 180,E1 -14116.271,E2 -14116.271} C_VEL
LIN {X 0,Y 339.338,Z 515.863,A -85,B 0,C 180,E1 -14119.257,E2 -14119.257} C_VEL
LIN {X 0,Y 339.246,Z 519.916,A -85,B 0,C 180,E1 -14121.661,E2 -14121.661} C_VEL
LIN {X 0,Y 339.344,Z 522.902,A -85,B 0,C 180,E1 -14124.055,E2 -14124.055} C_VEL
LIN {X 0,Y 339.319,Z 524.719,A -85,B 0,C 180,E1 -14126.437,E2 -14126.437} C_VEL
LIN {X 0,Y 339.488,Z 525.217,A -85,B 0,C 180,E1 -14127.626,E2 -14127.626} C_VEL
LIN {X 0,Y 339.578,Z 525.404,A -85,B 0,C 180,E1 -14129.999,E2 -14129.999} C_VEL
LIN {X 0,Y 339.521,Z 524.362,A -85,B 0,C 180,E1 -14132.372,E2 -14132.372} C_VEL
LIN {X 0,Y 339.369,Z 522.192,A -85,B 0,C 180,E1 -14134.751,E2 -14134.751} C_VEL
LIN {X 0,Y 339.462,Z 519.982,A -85,B 0,C 180,E1 -14136.407,E2 -14136.407} C_VEL
LIN {X 0,Y 339.365,Z 515.488,A -85,B 0,C 180,E1 -14138.934,E2 -14138.934} C_VEL
LIN {X 0,Y 339.529,Z 509.858,A -85,B 0,C 180,E1 -14141.34,E2 -14141.34} C_VEL
LIN {X 0,Y 340.029,Z 502.304,A -85,B 0,C 180,E1 -14143.91,E2 -14143.91} C_VEL
LIN {X 0,Y 340.689,Z 494.212,A -85,B 0,C 180,E1 -14146.169,E2 -14146.169} C_VEL
LIN {X 0,Y 341.706,Z 484.158,A -85,B 0,C 180,E1 -14148.518,E2 -14148.518} C_VEL
LIN {X 0,Y 343.05,Z 473.073,A -85,B 0,C 180,E1 -14150.694,E2 -14150.694} C_VEL
LIN {X 0,Y 344.456,Z 462.312,A -85,B 0,C 180,E1 -14152.491,E2 -14152.491} C_VEL
LIN {X 0,Y 346.196,Z 449.838,A -85,B 0,C 180,E1 -14154.272,E2 -14154.272} C_VEL
LIN {X 0,Y 347.936,Z 436.481,A -85,B 0,C 180,E1 -14155.899,E2 -14155.899} C_VEL
LIN {X 0,Y 349.824,Z 422.282,A -85,B 0,C 180,E1 -14157.358,E2 -14157.358} C_VEL
LIN {X 0,Y 351.74,Z 407.127,A -85,B 0,C 180,E1 -14158.654,E2 -14158.654} C_VEL
LIN {X 0,Y 353.589,Z 390.68,A -85,B 0,C 180,E1 -14159.794,E2 -14159.794} C_VEL
LIN {X 0,Y 355.389,Z 372.447,A -85,B 0,C 180,E1 -14160.776,E2 -14160.776} C_VEL
LIN {X 0,Y 356.795,Z 354.914,A -85,B 0,C 180,E1 -14161.465,E2 -14161.465} C_VEL
LIN {X 0,Y 364.825,Z 195.733,A -85,B 0,C 180,E1 -14165.724,E2 -14165.724} C_VEL
LIN {X 0,Y 361.733,Z 169.434,A -85,B 0,C 180,E1 -14166.807,E2 -14166.807} C_VEL
LIN {X 0,Y 350.751,Z 144.945,A -85,B 0,C 180,E1 -14168.608,E2 -14168.608} C_VEL
LIN {X 0,Y 345.146,Z 127.572,A -85,B 0,C 180,E1 -14171.556,E2 -14171.556} C_VEL
LIN {X 0,Y 340.71,Z 114.359,A -85,B 0,C 180,E1 -14173.942,E2 -14173.942} C_VEL
LIN {X 0,Y 340.695,Z 114.358,A -85,B 0,C 180,E1 -14177.954,E2 -14177.954} C_VEL
LIN {X 0,Y 340.731,Z 114.353,A -85,B 0,C 180,E1 -14181.773,E2 -14181.773} C_VEL
LIN {X 0,Y 340.718,Z 114.354,A -85,B 0,C 180,E1 -14185.595,E2 -14185.595} C_VEL
LIN {X 0,Y 340.711,Z 114.354,A -85,B 0,C 180,E1 -14188.957,E2 -14188.957} C_VEL
LIN {X 0,Y 340.775,Z 114.348,A -85,B 0,C 180,E1 -14192.474,E2 -14192.474} C_VEL
LIN {X 0,Y 340.751,Z 114.351,A -85,B 0,C 180,E1 -14195.638,E2 -14195.638} C_VEL
LIN {X 0,Y 340.743,Z 114.351,A -85,B 0,C 180,E1 -14199.474,E2 -14199.474} C_VEL
LIN {X 0,Y 340.854,Z 114.342,A -85,B 0,C 180,E1 -14201.984,E2 -14201.984} C_VEL
LIN {X 0,Y 340.864,Z 114.339,A -85,B 0,C 180,E1 -14205.705,E2 -14205.705} C_VEL
LIN {X 0,Y 340.87,Z 114.335,A -85,B 0,C 180,E1 -14209.306,E2 -14209.306} C_VEL
LIN {X 0,Y 341.071,Z 114.309,A -85,B 0,C 180,E1 -14212.898,E2 -14212.898} C_VEL
LIN {X 0,Y 341.165,Z 114.303,A -85,B 0,C 180,E1 -14217.639,E2 -14217.639} C_VEL
LIN {X 0,Y 341.311,Z 114.281,A -85,B 0,C 180,E1 -14220,E2 -14220} C_VEL
LIN {X 0,Y 341.166,Z 114.297,A -85,B 0,C 180,E1 -14222.361,E2 -14222.361} C_VEL
LIN {X 0,Y 341.073,Z 114.311,A -85,B 0,C 180,E1 -14227.102,E2 -14227.102} C_VEL
LIN {X 0,Y 340.866,Z 114.335,A -85,B 0,C 180,E1 -14230.694,E2 -14230.694} C_VEL
LIN {X 0,Y 340.858,Z 114.335,A -85,B 0,C 180,E1 -14234.325,E2 -14234.325} C_VEL
LIN {X 0,Y 340.832,Z 114.339,A -85,B 0,C 180,E1 -14238.467,E2 -14238.467} C_VEL
LIN {X 0,Y 340.749,Z 114.35,A -85,B 0,C 180,E1 -14241.857,E2 -14241.857} C_VEL
LIN {X 0,Y 340.768,Z 114.348,A -85,B 0,C 180,E1 -14245.665,E2 -14245.665} C_VEL
LIN {X 0,Y 340.724,Z 114.352,A -85,B 0,C 180,E1 -14248.321,E2 -14248.321} C_VEL
LIN {X 0,Y 340.693,Z 114.362,A -85,B 0,C 180,E1 -14251.045,E2 -14251.045} C_VEL
LIN {X 0,Y 340.714,Z 114.357,A -85,B 0,C 180,E1 -14255.279,E2 -14255.279} C_VEL
LIN {X 0,Y 340.706,Z 114.355,A -85,B 0,C 180,E1 -14258.387,E2 -14258.387} C_VEL
LIN {X 0,Y 340.696,Z 114.356,A -85,B 0,C 180,E1 -14262.046,E2 -14262.046} C_VEL
LIN {X 0,Y 340.691,Z 114.357,A -85,B 0,C 180,E1 -14265.464,E2 -14265.464} C_VEL
LIN {X 0,Y 340.702,Z 114.36,A -85,B 0,C 180,E1 -14268.694,E2 -14268.694} C_VEL
LIN {X 0,Y 340.734,Z 114.351,A -85,B 0,C 180,E1 -14271.774,E2 -14271.774} C_VEL
LIN {X 0,Y 340.72,Z 114.353,A -85,B 0,C 180,E1 -14275.596,E2 -14275.596} C_VEL
LIN {X 0,Y 340.695,Z 114.358,A -85,B 0,C 180,E1 -14278.956,E2 -14278.956} C_VEL
LIN {X 0,Y 340.801,Z 114.344,A -85,B 0,C 180,E1 -14283.021,E2 -14283.021} C_VEL
LIN {X 0,Y 340.729,Z 114.353,A -85,B 0,C 180,E1 -14286.928,E2 -14286.928} C_VEL
LIN {X 0,Y 340.799,Z 114.346,A -85,B 0,C 180,E1 -14290.735,E2 -14290.735} C_VEL
LIN {X 0,Y 340.786,Z 114.344,A -85,B 0,C 180,E1 -14293.219,E2 -14293.219} C_VEL
LIN {X 0,Y 340.844,Z 114.338,A -85,B 0,C 180,E1 -14296.891,E2 -14296.891} C_VEL
LIN {X 0,Y 340.929,Z 114.33,A -85,B 0,C 180,E1 -14300.509,E2 -14300.509} C_VEL
LIN {X 0,Y 341.076,Z 114.309,A -85,B 0,C 180,E1 -14302.899,E2 -14302.899} C_VEL
LIN {X 0,Y 341.169,Z 114.299,A -85,B 0,C 180,E1 -14307.64,E2 -14307.64} C_VEL
LIN {X 0,Y 341.296,Z 114.286,A -85,B 0,C 180,E1 -14310.001,E2 -14310.001} C_VEL
LIN {X 0,Y 341.169,Z 114.299,A -85,B 0,C 180,E1 -14312.362,E2 -14312.362} C_VEL
LIN {X 0,Y 341.077,Z 114.308,A -85,B 0,C 180,E1 -14317.103,E2 -14317.103} C_VEL
LIN {X 0,Y 340.873,Z 114.334,A -85,B 0,C 180,E1 -14320.694,E2 -14320.694} C_VEL
LIN {X 0,Y 340.865,Z 114.336,A -85,B 0,C 180,E1 -14324.326,E2 -14324.326} C_VEL
LIN {X 0,Y 340.839,Z 114.338,A -85,B 0,C 180,E1 -14328.467,E2 -14328.467} C_VEL
LIN {X 0,Y 340.756,Z 114.352,A -85,B 0,C 180,E1 -14331.858,E2 -14331.858} C_VEL
LIN {X 0,Y 340.775,Z 114.351,A -85,B 0,C 180,E1 -14335.665,E2 -14335.665} C_VEL
LIN {X 0,Y 340.731,Z 114.352,A -85,B 0,C 180,E1 -14338.321,E2 -14338.321} C_VEL
LIN {X 0,Y 340.7,Z 114.357,A -85,B 0,C 180,E1 -14341.045,E2 -14341.045} C_VEL
LIN {X 0,Y 340.721,Z 114.357,A -85,B 0,C 180,E1 -14345.279,E2 -14345.279} C_VEL
LIN {X 0,Y 340.714,Z 114.353,A -85,B 0,C 180,E1 -14348.387,E2 -14348.387} C_VEL
LIN {X 0,Y 340.702,Z 114.355,A -85,B 0,C 180,E1 -14352.046,E2 -14352.046} C_VEL
LIN {X 0,Y 340.687,Z 114.361,A -85,B 0,C 180,E1 -14355.462,E2 -14355.462} C_VEL
LIN {X 0,Y 340.689,Z 114.358,A -85,B 0,C 180,E1 -14358.691,E2 -14358.691} C_VEL
LIN {X 0,Y 340.745,Z 114.473,A -85,B 0,C 180,E1 -14361.424,E2 -14361.424} C_VEL
LIN {X 0,Y 341.645,Z 117.052,A -85,B 0,C 180,E1 -14361.601,E2 -14361.601} C_VEL
LIN {X 0,Y 354.751,Z 142.443,A -85,B 0,C 180,E1 -14363.654,E2 -14363.654} C_VEL
LIN {X 0,Y 364.206,Z 161.707,A -85,B 0,C 180,E1 -14365.062,E2 -14365.062} C_VEL
LIN {X 0,Y 363.812,Z 168.986,A -85,B 0,C 180,E1 -14365.252,E2 -14365.252} C_VEL
LIN {X 0,Y 362.982,Z 174.784,A -85,B 0,C 180,E1 -14365.361,E2 -14365.361} C_VEL
LIN {X 0,Y 356.74,Z 193.617,A -85,B 0,C 180,E1 -14365.447,E2 -14365.447} C_VEL
LIN {X 0,Y 355.799,Z 199.42,A -85,B 0,C 180,E1 -14365.554,E2 -14365.554} C_VEL
LIN {X 0,Y 350.624,Z 302.434,A -85,B 0,C 180,E1 -14368.38,E2 -14368.38} C_VEL
LIN {X 0,Y 349.563,Z 319.463,A -85,B 0,C 180,E1 -14369.074,E2 -14369.074} C_VEL
LIN {X 0,Y 348.249,Z 335.726,A -85,B 0,C 180,E1 -14369.953,E2 -14369.953} C_VEL
LIN {X 0,Y 346.971,Z 349.925,A -85,B 0,C 180,E1 -14370.914,E2 -14370.914} C_VEL
LIN {X 0,Y 345.19,Z 366.152,A -85,B 0,C 180,E1 -14372.242,E2 -14372.242} C_VEL
LIN {X 0,Y 343.346,Z 381.137,A -85,B 0,C 180,E1 -14373.727,E2 -14373.727} C_VEL
LIN {X 0,Y 341.501,Z 395.306,A -85,B 0,C 180,E1 -14375.404,E2 -14375.404} C_VEL
LIN {X 0,Y 339.794,Z 407.983,A -85,B 0,C 180,E1 -14377.182,E2 -14377.182} C_VEL
LIN {X 0,Y 338.213,Z 419.057,A -85,B 0,C 180,E1 -14378.995,E2 -14378.995} C_VEL
LIN {X 0,Y 336.805,Z 430.207,A -85,B 0,C 180,E1 -14381.129,E2 -14381.129} C_VEL
LIN {X 0,Y 335.483,Z 439.735,A -85,B 0,C 180,E1 -14383.259,E2 -14383.259} C_VEL
LIN {X 0,Y 334.454,Z 448.898,A -85,B 0,C 180,E1 -14385.705,E2 -14385.705} C_VEL
LIN {X 0,Y 333.633,Z 455.551,A -85,B 0,C 180,E1 -14387.839,E2 -14387.839} C_VEL
LIN {X 0,Y 333.107,Z 461.909,A -85,B 0,C 180,E1 -14390.283,E2 -14390.283} C_VEL
LIN {X 0,Y 332.793,Z 467,A -85,B 0,C 180,E1 -14392.72,E2 -14392.72} C_VEL
LIN {X 0,Y 332.507,Z 470.848,A -85,B 0,C 180,E1 -14395.15,E2 -14395.15} C_VEL
LIN {X 0,Y 332.527,Z 473.644,A -85,B 0,C 180,E1 -14397.577,E2 -14397.577} C_VEL
LIN {X 0,Y 332.451,Z 475.354,A -85,B 0,C 180,E1 -14400,E2 -14400} C_VEL
LIN {X 0,Y 332.7,Z 476.017,A -85,B 0,C 180,E1 -14402.421,E2 -14402.421} C_VEL
LIN {X 0,Y 333.01,Z 475.698,A -85,B 0,C 180,E1 -14404.842,E2 -14404.842} C_VEL
LIN {X 0,Y 333.684,Z 473.583,A -85,B 0,C 180,E1 -14408.143,E2 -14408.143} C_VEL
LIN {X 0,Y 334.636,Z 470.321,A -85,B 0,C 180,E1 -14410.895,E2 -14410.895} C_VEL
LIN {X 0,Y 335.785,Z 466.29,A -85,B 0,C 180,E1 -14413.31,E2 -14413.31} C_VEL
LIN {X 0,Y 337.18,Z 461.209,A -85,B 0,C 180,E1 -14415.722,E2 -14415.722} C_VEL
LIN {X 0,Y 339.159,Z 454.846,A -85,B 0,C 180,E1 -14418.109,E2 -14418.109} C_VEL
LIN {X 0,Y 341.793,Z 446.102,A -85,B 0,C 180,E1 -14420.775,E2 -14420.775} C_VEL
LIN {X 0,Y 344.307,Z 437.948,A -85,B 0,C 180,E1 -14422.819,E2 -14422.819} C_VEL
LIN {X 0,Y 347.511,Z 427.081,A -85,B 0,C 180,E1 -14425.131,E2 -14425.131} C_VEL
LIN {X 0,Y 350.737,Z 415.949,A -85,B 0,C 180,E1 -14427.12,E2 -14427.12} C_VEL
LIN {X 0,Y 354.374,Z 403.241,A -85,B 0,C 180,E1 -14429.016,E2 -14429.016} C_VEL
LIN {X 0,Y 357.828,Z 389.985,A -85,B 0,C 180,E1 -14430.707,E2 -14430.707} C_VEL
LIN {X 0,Y 361.583,Z 374.847,A -85,B 0,C 180,E1 -14432.311,E2 -14432.311} C_VEL
LIN {X 0,Y 365.441,Z 357.766,A -85,B 0,C 180,E1 -14433.791,E2 -14433.791} C_VEL
LIN {X 0,Y 368.894,Z 340.616,A -85,B 0,C 180,E1 -14434.993,E2 -14434.993} C_VEL
LIN {X 0,Y 371.781,Z 324.17,A -85,B 0,C 180,E1 -14435.916,E2 -14435.916} C_VEL
LIN {X 0,Y 374.505,Z 306.206,A -85,B 0,C 180,E1 -14436.689,E2 -14436.689} C_VEL
LIN {X 0,Y 384.699,Z 245.818,A -85,B 0,C 180,E1 -14438.86,E2 -14438.86} C_VEL
LIN {X 0,Y 395.454,Z 191.305,A -85,B 0,C 180,E1 -14440.791,E2 -14440.791} C_VEL
LIN {X 0,Y 394.439,Z 189.565,A -85,B 0,C 180,E1 -14441.986,E2 -14441.986} C_VEL
LIN {X 0,Y 393.549,Z 189.314,A -85,B 0,C 180,E1 -14443.508,E2 -14443.508} C_VEL
LIN {X 0,Y 393.3,Z 191.114,A -85,B 0,C 180,E1 -14445.366,E2 -14445.366} C_VEL
LIN {X 0,Y 393.521,Z 193.126,A -85,B 0,C 180,E1 -14446.372,E2 -14446.372} C_VEL
LIN {X 0,Y 394.197,Z 197.723,A -85,B 0,C 180,E1 -14447.839,E2 -14447.839} C_VEL
LIN {X 0,Y 394.327,Z 198.957,A -85,B 0,C 180,E1 -14448.109,E2 -14448.109} C_VEL
LIN {X 0,Y 393.402,Z 205.43,A -85,B 0,C 180,E1 -14448.532,E2 -14448.532} C_VEL
LIN {X 0,Y 381.003,Z 273.22,A -85,B 0,C 180,E1 -14450.903,E2 -14450.903} C_VEL
LIN {X 0,Y 369.805,Z 345.927,A -85,B 0,C 180,E1 -14453.523,E2 -14453.523} C_VEL
LIN {X 0,Y 366.109,Z 365.236,A -85,B 0,C 180,E1 -14454.415,E2 -14454.415} C_VEL
LIN {X 0,Y 362.221,Z 382.676,A -85,B 0,C 180,E1 -14455.421,E2 -14455.421} C_VEL
LIN {X 0,Y 358.231,Z 399.801,A -85,B 0,C 180,E1 -14456.679,E2 -14456.679} C_VEL
LIN {X 0,Y 354.234,Z 415.945,A -85,B 0,C 180,E1 -14458.113,E2 -14458.113} C_VEL
LIN {X 0,Y 350.07,Z 432.33,A -85,B 0,C 180,E1 -14459.873,E2 -14459.873} C_VEL
LIN {X 0,Y 346.464,Z 446.479,A -85,B 0,C 180,E1 -14461.695,E2 -14461.695} C_VEL
LIN {X 0,Y 343.36,Z 458.89,A -85,B 0,C 180,E1 -14463.564,E2 -14463.564} C_VEL
LIN {X 0,Y 340.101,Z 472.105,A -85,B 0,C 180,E1 -14465.912,E2 -14465.912} C_VEL
LIN {X 0,Y 337.559,Z 483.384,A -85,B 0,C 180,E1 -14468.311,E2 -14468.311} C_VEL
LIN {X 0,Y 335.527,Z 493.029,A -85,B 0,C 180,E1 -14470.74,E2 -14470.74} C_VEL
LIN {X 0,Y 334.242,Z 500.298,A -85,B 0,C 180,E1 -14472.879,E2 -14472.879} C_VEL
LIN {X 0,Y 333.197,Z 507.3,A -85,B 0,C 180,E1 -14475.338,E2 -14475.338} C_VEL
LIN {X 0,Y 332.506,Z 513.061,A -85,B 0,C 180,E1 -14477.797,E2 -14477.797} C_VEL
LIN {X 0,Y 332.168,Z 517.696,A -85,B 0,C 180,E1 -14480.254,E2 -14480.254} C_VEL
LIN {X 0,Y 332.223,Z 521.103,A -85,B 0,C 180,E1 -14482.707,E2 -14482.707} C_VEL
LIN {X 0,Y 332.261,Z 523.468,A -85,B 0,C 180,E1 -14485.146,E2 -14485.146} C_VEL
LIN {X 0,Y 332.422,Z 524.647,A -85,B 0,C 180,E1 -14487.576,E2 -14487.576} C_VEL
LIN {X 0,Y 332.519,Z 524.74,A -85,B 0,C 180,E1 -14489.999,E2 -14489.999} C_VEL
LIN {X 0,Y 332.46,Z 523.655,A -85,B 0,C 180,E1 -14492.422,E2 -14492.422} C_VEL
LIN {X 0,Y 332.31,Z 521.375,A -85,B 0,C 180,E1 -14494.852,E2 -14494.852} C_VEL
LIN {X 0,Y 332.407,Z 519.278,A -85,B 0,C 180,E1 -14496.433,E2 -14496.433} C_VEL
LIN {X 0,Y 332.316,Z 515.734,A -85,B 0,C 180,E1 -14498.513,E2 -14498.513} C_VEL
LIN {X 0,Y 332.379,Z 510.301,A -85,B 0,C 180,E1 -14500.969,E2 -14500.969} C_VEL
LIN {X 0,Y 332.823,Z 503.527,A -85,B 0,C 180,E1 -14503.43,E2 -14503.43} C_VEL
LIN {X 0,Y 333.471,Z 495.208,A -85,B 0,C 180,E1 -14505.9,E2 -14505.9} C_VEL
LIN {X 0,Y 334.55,Z 485.147,A -85,B 0,C 180,E1 -14508.367,E2 -14508.367} C_VEL
LIN {X 0,Y 335.763,Z 474.624,A -85,B 0,C 180,E1 -14510.523,E2 -14510.523} C_VEL
LIN {X 0,Y 337.228,Z 464.169,A -85,B 0,C 180,E1 -14512.354,E2 -14512.354} C_VEL
LIN {X 0,Y 339.04,Z 451.156,A -85,B 0,C 180,E1 -14514.306,E2 -14514.306} C_VEL
LIN {X 0,Y 340.81,Z 437.957,A -85,B 0,C 180,E1 -14515.989,E2 -14515.989} C_VEL
LIN {X 0,Y 342.747,Z 424.101,A -85,B 0,C 180,E1 -14517.474,E2 -14517.474} C_VEL
LIN {X 0,Y 344.855,Z 407.662,A -85,B 0,C 180,E1 -14518.935,E2 -14518.935} C_VEL
LIN {X 0,Y 346.874,Z 390.228,A -85,B 0,C 180,E1 -14520.179,E2 -14520.179} C_VEL
LIN {X 0,Y 348.731,Z 372.093,A -85,B 0,C 180,E1 -14521.176,E2 -14521.176} C_VEL
LIN {X 0,Y 350.274,Z 353.714,A -85,B 0,C 180,E1 -14521.908,E2 -14521.908} C_VEL
LIN {X 0,Y 358.452,Z 196.453,A -85,B 0,C 180,E1 -14526.225,E2 -14526.225} C_VEL
LIN {X 0,Y 355.635,Z 172.102,A -85,B 0,C 180,E1 -14527.248,E2 -14527.248} C_VEL
LIN {X 0,Y 343.409,Z 144.648,A -85,B 0,C 180,E1 -14529.295,E2 -14529.295} C_VEL
LIN {X 0,Y 337.685,Z 127.124,A -85,B 0,C 180,E1 -14532.352,E2 -14532.352} C_VEL
LIN {X 0,Y 333.67,Z 115.236,A -85,B 0,C 180,E1 -14534.564,E2 -14534.564} C_VEL
LIN {X 0,Y 333.639,Z 115.236,A -85,B 0,C 180,E1 -14537.618,E2 -14537.618} C_VEL
LIN {X 0,Y 333.649,Z 115.234,A -85,B 0,C 180,E1 -14541.201,E2 -14541.201} C_VEL
LIN {X 0,Y 333.673,Z 115.233,A -85,B 0,C 180,E1 -14543.861,E2 -14543.861} C_VEL
LIN {X 0,Y 333.647,Z 115.234,A -85,B 0,C 180,E1 -14547.411,E2 -14547.411} C_VEL
LIN {X 0,Y 333.707,Z 115.227,A -85,B 0,C 180,E1 -14551.028,E2 -14551.028} C_VEL
LIN {X 0,Y 333.731,Z 115.226,A -85,B 0,C 180,E1 -14553.754,E2 -14553.754} C_VEL
LIN {X 0,Y 333.715,Z 115.23,A -85,B 0,C 180,E1 -14557.914,E2 -14557.914} C_VEL
LIN {X 0,Y 333.79,Z 115.219,A -85,B 0,C 180,E1 -14561.589,E2 -14561.589} C_VEL
LIN {X 0,Y 333.804,Z 115.217,A -85,B 0,C 180,E1 -14565.576,E2 -14565.576} C_VEL
LIN {X 0,Y 333.833,Z 115.211,A -85,B 0,C 180,E1 -14569.078,E2 -14569.078} C_VEL
LIN {X 0,Y 334.021,Z 115.187,A -85,B 0,C 180,E1 -14572.748,E2 -14572.748} C_VEL
LIN {X 0,Y 333.807,Z 115.214,A -85,B 0,C 180,E1 -14575.169,E2 -14575.169} C_VEL
LIN {X 0,Y 334.103,Z 115.182,A -85,B 0,C 180,E1 -14577.589,E2 -14577.589} C_VEL
LIN {X 0,Y 334.262,Z 115.16,A -85,B 0,C 180,E1 -14580,E2 -14580} C_VEL
LIN {X 0,Y 334.103,Z 115.177,A -85,B 0,C 180,E1 -14582.411,E2 -14582.411} C_VEL
LIN {X 0,Y 334.022,Z 115.19,A -85,B 0,C 180,E1 -14587.253,E2 -14587.253} C_VEL
LIN {X 0,Y 333.829,Z 115.212,A -85,B 0,C 180,E1 -14590.922,E2 -14590.922} C_VEL
LIN {X 0,Y 333.804,Z 115.215,A -85,B 0,C 180,E1 -14594.635,E2 -14594.635} C_VEL
LIN {X 0,Y 333.791,Z 115.216,A -85,B 0,C 180,E1 -14598.655,E2 -14598.655} C_VEL
LIN {X 0,Y 333.688,Z 115.229,A -85,B 0,C 180,E1 -14602.279,E2 -14602.279} C_VEL
LIN {X 0,Y 333.731,Z 115.223,A -85,B 0,C 180,E1 -14606.247,E2 -14606.247} C_VEL
LIN {X 0,Y 333.686,Z 115.233,A -85,B 0,C 180,E1 -14608.975,E2 -14608.975} C_VEL
LIN {X 0,Y 333.639,Z 115.236,A -85,B 0,C 180,E1 -14612.587,E2 -14612.587} C_VEL
LIN {X 0,Y 333.673,Z 115.231,A -85,B 0,C 180,E1 -14616.139,E2 -14616.139} C_VEL
LIN {X 0,Y 333.643,Z 115.237,A -85,B 0,C 180,E1 -14619.193,E2 -14619.193} C_VEL
LIN {X 0,Y 333.63,Z 115.238,A -85,B 0,C 180,E1 -14622.501,E2 -14622.501} C_VEL
LIN {X 0,Y 333.64,Z 115.234,A -85,B 0,C 180,E1 -14625.964,E2 -14625.964} C_VEL
LIN {X 0,Y 333.653,Z 115.234,A -85,B 0,C 180,E1 -14629.314,E2 -14629.314} C_VEL
LIN {X 0,Y 333.652,Z 115.235,A -85,B 0,C 180,E1 -14632.35,E2 -14632.35} C_VEL
LIN {X 0,Y 333.671,Z 115.231,A -85,B 0,C 180,E1 -14635.342,E2 -14635.342} C_VEL
LIN {X 0,Y 333.688,Z 115.229,A -85,B 0,C 180,E1 -14639.638,E2 -14639.638} C_VEL
LIN {X 0,Y 333.738,Z 115.226,A -85,B 0,C 180,E1 -14642.402,E2 -14642.402} C_VEL
LIN {X 0,Y 333.725,Z 115.225,A -85,B 0,C 180,E1 -14645.092,E2 -14645.092} C_VEL
LIN {X 0,Y 333.692,Z 115.229,A -85,B 0,C 180,E1 -14649.021,E2 -14649.021} C_VEL
LIN {X 0,Y 333.794,Z 115.216,A -85,B 0,C 180,E1 -14651.59,E2 -14651.59} C_VEL
LIN {X 0,Y 333.808,Z 115.214,A -85,B 0,C 180,E1 -14655.577,E2 -14655.577} C_VEL
LIN {X 0,Y 333.834,Z 115.211,A -85,B 0,C 180,E1 -14659.079,E2 -14659.079} C_VEL
LIN {X 0,Y 334.026,Z 115.188,A -85,B 0,C 180,E1 -14662.748,E2 -14662.748} C_VEL
LIN {X 0,Y 333.81,Z 115.213,A -85,B 0,C 180,E1 -14665.17,E2 -14665.17} C_VEL
LIN {X 0,Y 334.106,Z 115.178,A -85,B 0,C 180,E1 -14667.59,E2 -14667.59} C_VEL
LIN {X 0,Y 334.246,Z 115.165,A -85,B 0,C 180,E1 -14670.001,E2 -14670.001} C_VEL
LIN {X 0,Y 334.106,Z 115.178,A -85,B 0,C 180,E1 -14672.412,E2 -14672.412} C_VEL
LIN {X 0,Y 334.027,Z 115.187,A -85,B 0,C 180,E1 -14677.253,E2 -14677.253} C_VEL
LIN {X 0,Y 333.835,Z 115.21,A -85,B 0,C 180,E1 -14680.923,E2 -14680.923} C_VEL
LIN {X 0,Y 333.81,Z 115.214,A -85,B 0,C 180,E1 -14684.635,E2 -14684.635} C_VEL
LIN {X 0,Y 333.798,Z 115.215,A -85,B 0,C 180,E1 -14688.656,E2 -14688.656} C_VEL
LIN {X 0,Y 333.695,Z 115.229,A -85,B 0,C 180,E1 -14692.279,E2 -14692.279} C_VEL
LIN {X 0,Y 333.737,Z 115.223,A -85,B 0,C 180,E1 -14696.247,E2 -14696.247} C_VEL
LIN {X 0,Y 333.692,Z 115.229,A -85,B 0,C 180,E1 -14698.975,E2 -14698.975} C_VEL
LIN {X 0,Y 333.646,Z 115.234,A -85,B 0,C 180,E1 -14702.588,E2 -14702.588} C_VEL
LIN {X 0,Y 333.679,Z 115.23,A -85,B 0,C 180,E1 -14706.139,E2 -14706.139} C_VEL
LIN {X 0,Y 333.65,Z 115.238,A -85,B 0,C 180,E1 -14709.193,E2 -14709.193} C_VEL
LIN {X 0,Y 333.636,Z 115.235,A -85,B 0,C 180,E1 -14712.501,E2 -14712.501} C_VEL
LIN {X 0,Y 333.625,Z 115.237,A -85,B 0,C 180,E1 -14715.96,E2 -14715.96} C_VEL
LIN {X 0,Y 333.65,Z 115.238,A -85,B 0,C 180,E1 -14719.316,E2 -14719.316} C_VEL
LIN {X 0,Y 333.681,Z 115.232,A -85,B 0,C 180,E1 -14720.74,E2 -14720.74} C_VEL
LIN {X 0,Y 334.766,Z 118.195,A -85,B 0,C 180,E1 -14720.967,E2 -14720.967} C_VEL
LIN {X 0,Y 348.946,Z 145.749,A -85,B 0,C 180,E1 -14723.251,E2 -14723.251} C_VEL
LIN {X 0,Y 357.797,Z 163.751,A -85,B 0,C 180,E1 -14724.594,E2 -14724.594} C_VEL
LIN {X 0,Y 355.799,Z 199.42,A -85,B 0,C 180,E1 -14725.554,E2 -14725.554} C_VEL
LIN {X 0,Y 354.878,Z 205.217,A -85,B 0,C 180,E1 -14725.663,E2 -14725.663} C_VEL
LIN {X 0,Y 348.695,Z 224.053,A -85,B 0,C 180,E1 -14725.782,E2 -14725.782} C_VEL
LIN {X 0,Y 347.766,Z 229.851,A -85,B 0,C 180,E1 -14725.895,E2 -14725.895} C_VEL
LIN {X 0,Y 344.001,Z 302.898,A -85,B 0,C 180,E1 -14727.958,E2 -14727.958} C_VEL
LIN {X 0,Y 342.786,Z 321.349,A -85,B 0,C 180,E1 -14728.737,E2 -14728.737} C_VEL
LIN {X 0,Y 341.31,Z 338.98,A -85,B 0,C 180,E1 -14729.74,E2 -14729.74} C_VEL
LIN {X 0,Y 339.742,Z 355.188,A -85,B 0,C 180,E1 -14730.914,E2 -14730.914} C_VEL
LIN {X 0,Y 337.933,Z 370.525,A -85,B 0,C 180,E1 -14732.268,E2 -14732.268} C_VEL
LIN {X 0,Y 336.043,Z 384.841,A -85,B 0,C 180,E1 -14733.781,E2 -14733.781} C_VEL
LIN {X 0,Y 334.132,Z 399.406,A -85,B 0,C 180,E1 -14735.62,E2 -14735.62} C_VEL
LIN {X 0,Y 332.245,Z 412.734,A -85,B 0,C 180,E1 -14737.619,E2 -14737.619} C_VEL
LIN {X 0,Y 330.689,Z 423.995,A -85,B 0,C 180,E1 -14739.606,E2 -14739.606} C_VEL
LIN {X 0,Y 329.314,Z 433.953,A -85,B 0,C 180,E1 -14741.652,E2 -14741.652} C_VEL
LIN {X 0,Y 327.98,Z 444.128,A -85,B 0,C 180,E1 -14744.135,E2 -14744.135} C_VEL
LIN {X 0,Y 327.086,Z 451.661,A -85,B 0,C 180,E1 -14746.328,E2 -14746.328} C_VEL
LIN {X 0,Y 326.321,Z 458.867,A -85,B 0,C 180,E1 -14748.823,E2 -14748.823} C_VEL
LIN {X 0,Y 325.865,Z 464.729,A -85,B 0,C 180,E1 -14751.317,E2 -14751.317} C_VEL
LIN {X 0,Y 325.554,Z 469.274,A -85,B 0,C 180,E1 -14753.803,E2 -14753.803} C_VEL
LIN {X 0,Y 325.409,Z 472.728,A -85,B 0,C 180,E1 -14756.285,E2 -14756.285} C_VEL
LIN {X 0,Y 325.466,Z 474.064,A -85,B 0,C 180,E1 -14757.525,E2 -14757.525} C_VEL
LIN {X 0,Y 325.384,Z 475.853,A -85,B 0,C 180,E1 -14760,E2 -14760} C_VEL
LIN {X 0,Y 325.639,Z 476.651,A -85,B 0,C 180,E1 -14762.474,E2 -14762.474} C_VEL
LIN {X 0,Y 325.981,Z 476.406,A -85,B 0,C 180,E1 -14764.947,E2 -14764.947} C_VEL
LIN {X 0,Y 326.333,Z 475.155,A -85,B 0,C 180,E1 -14767.424,E2 -14767.424} C_VEL
LIN {X 0,Y 327.267,Z 472.89,A -85,B 0,C 180,E1 -14769.892,E2 -14769.892} C_VEL
LIN {X 0,Y 328.643,Z 468.56,A -85,B 0,C 180,E1 -14772.976,E2 -14772.976} C_VEL
LIN {X 0,Y 330.464,Z 462.539,A -85,B 0,C 180,E1 -14776.05,E2 -14776.05} C_VEL
LIN {X 0,Y 332.575,Z 456.307,A -85,B 0,C 180,E1 -14778.48,E2 -14778.48} C_VEL
LIN {X 0,Y 335.033,Z 448.824,A -85,B 0,C 180,E1 -14780.892,E2 -14780.892} C_VEL
LIN {X 0,Y 338.045,Z 439.886,A -85,B 0,C 180,E1 -14783.267,E2 -14783.267} C_VEL
LIN {X 0,Y 341.423,Z 429.343,A -85,B 0,C 180,E1 -14785.612,E2 -14785.612} C_VEL
LIN {X 0,Y 344.837,Z 418.574,A -85,B 0,C 180,E1 -14787.623,E2 -14787.623} C_VEL
LIN {X 0,Y 349.011,Z 405.081,A -85,B 0,C 180,E1 -14789.711,E2 -14789.711} C_VEL
LIN {X 0,Y 352.596,Z 392.42,A -85,B 0,C 180,E1 -14791.381,E2 -14791.381} C_VEL
LIN {X 0,Y 356.921,Z 376.511,A -85,B 0,C 180,E1 -14793.121,E2 -14793.121} C_VEL
LIN {X 0,Y 361.127,Z 359.479,A -85,B 0,C 180,E1 -14794.638,E2 -14794.638} C_VEL
LIN {X 0,Y 365.094,Z 341.473,A -85,B 0,C 180,E1 -14795.927,E2 -14795.927} C_VEL
LIN {X 0,Y 368.488,Z 323.74,A -85,B 0,C 180,E1 -14796.926,E2 -14796.926} C_VEL
LIN {X 0,Y 372.039,Z 302.308,A -85,B 0,C 180,E1 -14797.832,E2 -14797.832} C_VEL
LIN {X 0,Y 383.676,Z 240.152,A -85,B 0,C 180,E1 -14800.089,E2 -14800.089} C_VEL
LIN {X 0,Y 392.883,Z 197.002,A -85,B 0,C 180,E1 -14801.619,E2 -14801.619} C_VEL
LIN {X 0,Y 392.538,Z 196.312,A -85,B 0,C 180,E1 -14802.14,E2 -14802.14} C_VEL
LIN {X 0,Y 391.737,Z 196.24,A -85,B 0,C 180,E1 -14803.552,E2 -14803.552} C_VEL
LIN {X 0,Y 391.456,Z 197.963,A -85,B 0,C 180,E1 -14805.244,E2 -14805.244} C_VEL
LIN {X 0,Y 391.54,Z 199.616,A -85,B 0,C 180,E1 -14806.058,E2 -14806.058} C_VEL
LIN {X 0,Y 391.929,Z 203.447,A -85,B 0,C 180,E1 -14807.324,E2 -14807.324} C_VEL
LIN {X 0,Y 391.323,Z 207.109,A -85,B 0,C 180,E1 -14807.568,E2 -14807.568} C_VEL
LIN {X 0,Y 378.298,Z 273.141,A -85,B 0,C 180,E1 -14809.899,E2 -14809.899} C_VEL
LIN {X 0,Y 366.175,Z 345.067,A -85,B 0,C 180,E1 -14812.541,E2 -14812.541} C_VEL
LIN {X 0,Y 362.144,Z 364.424,A -85,B 0,C 180,E1 -14813.448,E2 -14813.448} C_VEL
LIN {X 0,Y 358.064,Z 381.457,A -85,B 0,C 180,E1 -14814.445,E2 -14814.445} C_VEL
LIN {X 0,Y 354.222,Z 396.779,A -85,B 0,C 180,E1 -14815.565,E2 -14815.565} C_VEL
LIN {X 0,Y 349.939,Z 412.982,A -85,B 0,C 180,E1 -14816.991,E2 -14816.991} C_VEL
LIN {X 0,Y 345.642,Z 428.64,A -85,B 0,C 180,E1 -14818.648,E2 -14818.648} C_VEL
LIN {X 0,Y 341.745,Z 442.742,A -85,B 0,C 180,E1 -14820.424,E2 -14820.424} C_VEL
LIN {X 0,Y 338.019,Z 456.238,A -85,B 0,C 180,E1 -14822.443,E2 -14822.443} C_VEL
LIN {X 0,Y 334.507,Z 469.335,A -85,B 0,C 180,E1 -14824.766,E2 -14824.766} C_VEL
LIN {X 0,Y 331.549,Z 481.066,A -85,B 0,C 180,E1 -14827.24,E2 -14827.24} C_VEL
LIN {X 0,Y 329.269,Z 490.913,A -85,B 0,C 180,E1 -14829.705,E2 -14829.705} C_VEL
LIN {X 0,Y 327.741,Z 498.361,A -85,B 0,C 180,E1 -14831.884,E2 -14831.884} C_VEL
LIN {X 0,Y 326.447,Z 505.534,A -85,B 0,C 180,E1 -14834.388,E2 -14834.388} C_VEL
LIN {X 0,Y 325.665,Z 511.533,A -85,B 0,C 180,E1 -14836.903,E2 -14836.903} C_VEL
LIN {X 0,Y 325.144,Z 516.295,A -85,B 0,C 180,E1 -14839.412,E2 -14839.412} C_VEL
LIN {X 0,Y 325.07,Z 519.159,A -85,B 0,C 180,E1 -14841.295,E2 -14841.295} C_VEL
LIN {X 0,Y 325.191,Z 521.939,A -85,B 0,C 180,E1 -14843.796,E2 -14843.796} C_VEL
LIN {X 0,Y 325.154,Z 523.671,A -85,B 0,C 180,E1 -14846.281,E2 -14846.281} C_VEL
LIN {X 0,Y 325.336,Z 524.077,A -85,B 0,C 180,E1 -14847.523,E2 -14847.523} C_VEL
LIN {X 0,Y 325.461,Z 524.071,A -85,B 0,C 180,E1 -14849.999,E2 -14849.999} C_VEL
LIN {X 0,Y 325.4,Z 522.935,A -85,B 0,C 180,E1 -14852.475,E2 -14852.475} C_VEL
LIN {X 0,Y 325.254,Z 520.544,A -85,B 0,C 180,E1 -14854.957,E2 -14854.957} C_VEL
LIN {X 0,Y 325.344,Z 518.573,A -85,B 0,C 180,E1 -14856.448,E2 -14856.448} C_VEL
LIN {X 0,Y 325.237,Z 514.774,A -85,B 0,C 180,E1 -14858.699,E2 -14858.699} C_VEL
LIN {X 0,Y 325.34,Z 509.212,A -85,B 0,C 180,E1 -14861.21,E2 -14861.21} C_VEL
LIN {X 0,Y 325.818,Z 502.281,A -85,B 0,C 180,E1 -14863.725,E2 -14863.725} C_VEL
LIN {X 0,Y 326.513,Z 493.785,A -85,B 0,C 180,E1 -14866.248,E2 -14866.248} C_VEL
LIN {X 0,Y 327.473,Z 484.945,A -85,B 0,C 180,E1 -14868.454,E2 -14868.454} C_VEL
LIN {X 0,Y 328.709,Z 474.456,A -85,B 0,C 180,E1 -14870.657,E2 -14870.657} C_VEL
LIN {X 0,Y 330.212,Z 464.061,A -85,B 0,C 180,E1 -14872.525,E2 -14872.525} C_VEL
LIN {X 0,Y 331.992,Z 451.551,A -85,B 0,C 180,E1 -14874.457,E2 -14874.457} C_VEL
LIN {X 0,Y 333.867,Z 437.998,A -85,B 0,C 180,E1 -14876.234,E2 -14876.234} C_VEL
LIN {X 0,Y 336.023,Z 422.717,A -85,B 0,C 180,E1 -14877.902,E2 -14877.902} C_VEL
LIN {X 0,Y 338.16,Z 406.802,A -85,B 0,C 180,E1 -14879.33,E2 -14879.33} C_VEL
LIN {X 0,Y 340.18,Z 389.567,A -85,B 0,C 180,E1 -14880.579,E2 -14880.579} C_VEL
LIN {X 0,Y 342.106,Z 371.449,A -85,B 0,C 180,E1 -14881.59,E2 -14881.59} C_VEL
LIN {X 0,Y 343.673,Z 353.144,A -85,B 0,C 180,E1 -14882.335,E2 -14882.335} C_VEL
LIN {X 0,Y 352.122,Z 197.271,A -85,B 0,C 180,E1 -14886.732,E2 -14886.732} C_VEL
LIN {X 0,Y 349.49,Z 174.548,A -85,B 0,C 180,E1 -14887.711,E2 -14887.711} C_VEL
LIN {X 0,Y 337.116,Z 146.911,A -85,B 0,C 180,E1 -14889.817,E2 -14889.817} C_VEL
LIN {X 0,Y 335.842,Z 143.911,A -85,B 0,C 180,E1 -14890.083,E2 -14890.083} C_VEL
LIN {X 0,Y 330.235,Z 126.965,A -85,B 0,C 180,E1 -14893.13,E2 -14893.13} C_VEL
LIN {X 0,Y 326.604,Z 116.116,A -85,B 0,C 180,E1 -14895.197,E2 -14895.197} C_VEL
LIN {X 0,Y 326.574,Z 116.117,A -85,B 0,C 180,E1 -14898.868,E2 -14898.868} C_VEL
LIN {X 0,Y 326.625,Z 116.11,A -85,B 0,C 180,E1 -14902.761,E2 -14902.761} C_VEL
LIN {X 0,Y 326.604,Z 116.115,A -85,B 0,C 180,E1 -14905.981,E2 -14905.981} C_VEL
LIN {X 0,Y 326.637,Z 116.108,A -85,B 0,C 180,E1 -14909.388,E2 -14909.388} C_VEL
LIN {X 0,Y 326.681,Z 116.102,A -85,B 0,C 180,E1 -14913.142,E2 -14913.142} C_VEL
LIN {X 0,Y 326.647,Z 116.11,A -85,B 0,C 180,E1 -14915.871,E2 -14915.871} C_VEL
LIN {X 0,Y 326.66,Z 116.109,A -85,B 0,C 180,E1 -14919.865,E2 -14919.865} C_VEL
LIN {X 0,Y 326.696,Z 116.101,A -85,B 0,C 180,E1 -14922.472,E2 -14922.472} C_VEL
LIN {X 0,Y 326.756,Z 116.094,A -85,B 0,C 180,E1 -14926.315,E2 -14926.315} C_VEL
LIN {X 0,Y 326.811,Z 116.089,A -85,B 0,C 180,E1 -14930.094,E2 -14930.094} C_VEL
LIN {X 0,Y 326.975,Z 116.065,A -85,B 0,C 180,E1 -14932.59,E2 -14932.59} C_VEL
LIN {X 0,Y 326.774,Z 116.089,A -85,B 0,C 180,E1 -14935.065,E2 -14935.065} C_VEL
LIN {X 0,Y 327.043,Z 116.06,A -85,B 0,C 180,E1 -14937.537,E2 -14937.537} C_VEL
LIN {X 0,Y 327.212,Z 116.038,A -85,B 0,C 180,E1 -14940,E2 -14940} C_VEL
LIN {X 0,Y 327.044,Z 116.056,A -85,B 0,C 180,E1 -14942.463,E2 -14942.463} C_VEL
LIN {X 0,Y 326.966,Z 116.066,A -85,B 0,C 180,E1 -14946.665,E2 -14946.665} C_VEL
LIN {X 0,Y 326.809,Z 116.087,A -85,B 0,C 180,E1 -14949.907,E2 -14949.907} C_VEL
LIN {X 0,Y 326.755,Z 116.095,A -85,B 0,C 180,E1 -14953.686,E2 -14953.686} C_VEL
LIN {X 0,Y 326.695,Z 116.103,A -85,B 0,C 180,E1 -14957.528,E2 -14957.528} C_VEL
LIN {X 0,Y 326.661,Z 116.104,A -85,B 0,C 180,E1 -14960.135,E2 -14960.135} C_VEL
LIN {X 0,Y 326.648,Z 116.105,A -85,B 0,C 180,E1 -14964.129,E2 -14964.129} C_VEL
LIN {X 0,Y 326.679,Z 116.105,A -85,B 0,C 180,E1 -14966.858,E2 -14966.858} C_VEL
LIN {X 0,Y 326.63,Z 116.109,A -85,B 0,C 180,E1 -14970.61,E2 -14970.61} C_VEL
LIN {X 0,Y 326.603,Z 116.111,A -85,B 0,C 180,E1 -14974.02,E2 -14974.02} C_VEL
LIN {X 0,Y 326.624,Z 116.111,A -85,B 0,C 180,E1 -14977.239,E2 -14977.239} C_VEL
LIN {X 0,Y 326.574,Z 116.118,A -85,B 0,C 180,E1 -14981.132,E2 -14981.132} C_VEL
LIN {X 0,Y 326.56,Z 116.121,A -85,B 0,C 180,E1 -14984.75,E2 -14984.75} C_VEL
LIN {X 0,Y 326.599,Z 116.112,A -85,B 0,C 180,E1 -14988.159,E2 -14988.159} C_VEL
LIN {X 0,Y 326.638,Z 116.107,A -85,B 0,C 180,E1 -14991.395,E2 -14991.395} C_VEL
LIN {X 0,Y 326.617,Z 116.113,A -85,B 0,C 180,E1 -14994.852,E2 -14994.852} C_VEL
LIN {X 0,Y 326.605,Z 116.111,A -85,B 0,C 180,E1 -14997.456,E2 -14997.456} C_VEL
LIN {X 0,Y 326.645,Z 116.109,A -85,B 0,C 180,E1 -15000.34,E2 -15000.34} C_VEL
LIN {X 0,Y 326.688,Z 116.106,A -85,B 0,C 180,E1 -15004.517,E2 -15004.517} C_VEL
LIN {X 0,Y 326.652,Z 116.109,A -85,B 0,C 180,E1 -15008.547,E2 -15008.547} C_VEL
LIN {X 0,Y 326.743,Z 116.094,A -85,B 0,C 180,E1 -15011.178,E2 -15011.178} C_VEL
LIN {X 0,Y 326.762,Z 116.091,A -85,B 0,C 180,E1 -15015.434,E2 -15015.434} C_VEL
LIN {X 0,Y 326.77,Z 116.091,A -85,B 0,C 180,E1 -15018.84,E2 -15018.84} C_VEL
LIN {X 0,Y 326.98,Z 116.066,A -85,B 0,C 180,E1 -15022.591,E2 -15022.591} C_VEL
LIN {X 0,Y 326.777,Z 116.089,A -85,B 0,C 180,E1 -15025.066,E2 -15025.066} C_VEL
LIN {X 0,Y 327.047,Z 116.057,A -85,B 0,C 180,E1 -15027.538,E2 -15027.538} C_VEL
LIN {X 0,Y 327.198,Z 116.043,A -85,B 0,C 180,E1 -15030.001,E2 -15030.001} C_VEL
LIN {X 0,Y 327.047,Z 116.057,A -85,B 0,C 180,E1 -15032.464,E2 -15032.464} C_VEL
LIN {X 0,Y 326.997,Z 116.066,A -85,B 0,C 180,E1 -15036.17,E2 -15036.17} C_VEL
LIN {X 0,Y 326.916,Z 116.073,A -85,B 0,C 180,E1 -15038.656,E2 -15038.656} C_VEL
LIN {X 0,Y 326.736,Z 116.095,A -85,B 0,C 180,E1 -15042.422,E2 -15042.422} C_VEL
LIN {X 0,Y 326.756,Z 116.093,A -85,B 0,C 180,E1 -15044.958,E2 -15044.958} C_VEL
LIN {X 0,Y 326.734,Z 116.094,A -85,B 0,C 180,E1 -15048.839,E2 -15048.839} C_VEL
LIN {X 0,Y 326.623,Z 116.108,A -85,B 0,C 180,E1 -15052.788,E2 -15052.788} C_VEL
LIN {X 0,Y 326.692,Z 116.105,A -85,B 0,C 180,E1 -15055.484,E2 -15055.484} C_VEL
LIN {X 0,Y 326.65,Z 116.11,A -85,B 0,C 180,E1 -15059.661,E2 -15059.661} C_VEL
LIN {X 0,Y 326.609,Z 116.112,A -85,B 0,C 180,E1 -15064.02,E2 -15064.02} C_VEL
LIN {X 0,Y 326.632,Z 116.112,A -85,B 0,C 180,E1 -15067.239,E2 -15067.239} C_VEL
LIN {X 0,Y 326.581,Z 116.118,A -85,B 0,C 180,E1 -15071.132,E2 -15071.132} C_VEL
LIN {X 0,Y 326.559,Z 116.119,A -85,B 0,C 180,E1 -15074.748,E2 -15074.748} C_VEL
LIN {X 0,Y 326.58,Z 116.115,A -85,B 0,C 180,E1 -15078.155,E2 -15078.155} C_VEL
LIN {X 0,Y 326.631,Z 116.211,A -85,B 0,C 180,E1 -15080.075,E2 -15080.075} C_VEL
LIN {X 0,Y 327.64,Z 118.999,A -85,B 0,C 180,E1 -15080.283,E2 -15080.283} C_VEL
LIN {X 0,Y 340.886,Z 144.544,A -85,B 0,C 180,E1 -15082.478,E2 -15082.478} C_VEL
LIN {X 0,Y 351.329,Z 165.717,A -85,B 0,C 180,E1 -15084.114,E2 -15084.114} C_VEL
LIN {X 0,Y 347.766,Z 229.851,A -85,B 0,C 180,E1 -15085.895,E2 -15085.895} C_VEL
LIN {X 0,Y 346.836,Z 235.643,A -85,B 0,C 180,E1 -15086.007,E2 -15086.007} C_VEL
LIN {X 0,Y 340.623,Z 254.452,A -85,B 0,C 180,E1 -15086.149,E2 -15086.149} C_VEL
LIN {X 0,Y 339.65,Z 260.244,A -85,B 0,C 180,E1 -15086.268,E2 -15086.268} C_VEL
LIN {X 0,Y 337.325,Z 303.945,A -85,B 0,C 180,E1 -15087.555,E2 -15087.555} C_VEL
LIN {X 0,Y 336.158,Z 321.485,A -85,B 0,C 180,E1 -15088.313,E2 -15088.313} C_VEL
LIN {X 0,Y 334.605,Z 339.529,A -85,B 0,C 180,E1 -15089.36,E2 -15089.36} C_VEL
LIN {X 0,Y 332.924,Z 356.348,A -85,B 0,C 180,E1 -15090.606,E2 -15090.606} C_VEL
LIN {X 0,Y 330.874,Z 373.14,A -85,B 0,C 180,E1 -15092.141,E2 -15092.141} C_VEL
LIN {X 0,Y 328.821,Z 388.575,A -85,B 0,C 180,E1 -15093.856,E2 -15093.856} C_VEL
LIN {X 0,Y 326.843,Z 402.561,A -85,B 0,C 180,E1 -15095.717,E2 -15095.717} C_VEL
LIN {X 0,Y 324.95,Z 415.487,A -85,B 0,C 180,E1 -15097.76,E2 -15097.76} C_VEL
LIN {X 0,Y 323.38,Z 427.351,A -85,B 0,C 180,E1 -15099.983,E2 -15099.983} C_VEL
LIN {X 0,Y 321.869,Z 437.431,A -85,B 0,C 180,E1 -15102.2,E2 -15102.2} C_VEL
LIN {X 0,Y 320.654,Z 447.185,A -85,B 0,C 180,E1 -15104.751,E2 -15104.751} C_VEL
LIN {X 0,Y 319.664,Z 455.298,A -85,B 0,C 180,E1 -15107.299,E2 -15107.299} C_VEL
LIN {X 0,Y 319.014,Z 461.964,A -85,B 0,C 180,E1 -15109.849,E2 -15109.849} C_VEL
LIN {X 0,Y 318.648,Z 467.264,A -85,B 0,C 180,E1 -15112.395,E2 -15112.395} C_VEL
LIN {X 0,Y 318.383,Z 471.407,A -85,B 0,C 180,E1 -15114.934,E2 -15114.934} C_VEL
LIN {X 0,Y 318.387,Z 474.43,A -85,B 0,C 180,E1 -15117.47,E2 -15117.47} C_VEL
LIN {X 0,Y 318.319,Z 476.347,A -85,B 0,C 180,E1 -15120,E2 -15120} C_VEL
LIN {X 0,Y 318.58,Z 477.288,A -85,B 0,C 180,E1 -15122.529,E2 -15122.529} C_VEL
LIN {X 0,Y 318.952,Z 477.123,A -85,B 0,C 180,E1 -15125.056,E2 -15125.056} C_VEL
LIN {X 0,Y 319.365,Z 476.019,A -85,B 0,C 180,E1 -15127.587,E2 -15127.587} C_VEL
LIN {X 0,Y 320.323,Z 473.845,A -85,B 0,C 180,E1 -15130.109,E2 -15130.109} C_VEL
LIN {X 0,Y 321.477,Z 470.633,A -85,B 0,C 180,E1 -15132.628,E2 -15132.628} C_VEL
LIN {X 0,Y 322.879,Z 466.43,A -85,B 0,C 180,E1 -15135.141,E2 -15135.141} C_VEL
LIN {X 0,Y 325.235,Z 459.996,A -85,B 0,C 180,E1 -15138.046,E2 -15138.046} C_VEL
LIN {X 0,Y 327.955,Z 452.52,A -85,B 0,C 180,E1 -15140.707,E2 -15140.707} C_VEL
LIN {X 0,Y 330.959,Z 444.195,A -85,B 0,C 180,E1 -15143.132,E2 -15143.132} C_VEL
LIN {X 0,Y 334.384,Z 434.615,A -85,B 0,C 180,E1 -15145.455,E2 -15145.455} C_VEL
LIN {X 0,Y 337.918,Z 424.35,A -85,B 0,C 180,E1 -15147.565,E2 -15147.565} C_VEL
LIN {X 0,Y 341.289,Z 414.495,A -85,B 0,C 180,E1 -15149.279,E2 -15149.279} C_VEL
LIN {X 0,Y 345.96,Z 399.947,A -85,B 0,C 180,E1 -15151.436,E2 -15151.436} C_VEL
LIN {X 0,Y 350.568,Z 384.749,A -85,B 0,C 180,E1 -15153.284,E2 -15153.284} C_VEL
LIN {X 0,Y 355.07,Z 368.876,A -85,B 0,C 180,E1 -15154.857,E2 -15154.857} C_VEL
LIN {X 0,Y 359.13,Z 353.2,A -85,B 0,C 180,E1 -15156.141,E2 -15156.141} C_VEL
LIN {X 0,Y 362.882,Z 336.794,A -85,B 0,C 180,E1 -15157.245,E2 -15157.245} C_VEL
LIN {X 0,Y 366.28,Z 319.802,A -85,B 0,C 180,E1 -15158.146,E2 -15158.146} C_VEL
LIN {X 0,Y 371.564,Z 291.02,A -85,B 0,C 180,E1 -15159.275,E2 -15159.275} C_VEL
LIN {X 0,Y 385.199,Z 226.121,A -85,B 0,C 180,E1 -15161.64,E2 -15161.64} C_VEL
LIN {X 0,Y 390.518,Z 203.085,A -85,B 0,C 180,E1 -15162.45,E2 -15162.45} C_VEL
LIN {X 0,Y 389.88,Z 203.272,A -85,B 0,C 180,E1 -15163.681,E2 -15163.681} C_VEL
LIN {X 0,Y 389.618,Z 204.925,A -85,B 0,C 180,E1 -15165.192,E2 -15165.192} C_VEL
LIN {X 0,Y 389.628,Z 206.786,A -85,B 0,C 180,E1 -15165.999,E2 -15165.999} C_VEL
LIN {X 0,Y 389.702,Z 208.518,A -85,B 0,C 180,E1 -15166.576,E2 -15166.576} C_VEL
LIN {X 0,Y 375.279,Z 276.747,A -85,B 0,C 180,E1 -15169,E2 -15169} C_VEL
LIN {X 0,Y 362.977,Z 343.756,A -85,B 0,C 180,E1 -15171.492,E2 -15171.492} C_VEL
LIN {X 0,Y 358.382,Z 364.272,A -85,B 0,C 180,E1 -15172.471,E2 -15172.471} C_VEL
LIN {X 0,Y 353.615,Z 382.655,A -85,B 0,C 180,E1 -15173.575,E2 -15173.575} C_VEL
LIN {X 0,Y 349.159,Z 398.876,A -85,B 0,C 180,E1 -15174.817,E2 -15174.817} C_VEL
LIN {X 0,Y 344.661,Z 414.391,A -85,B 0,C 180,E1 -15176.243,E2 -15176.243} C_VEL
LIN {X 0,Y 339.808,Z 430.67,A -85,B 0,C 180,E1 -15178.047,E2 -15178.047} C_VEL
LIN {X 0,Y 335.724,Z 444.215,A -85,B 0,C 180,E1 -15179.839,E2 -15179.839} C_VEL
LIN {X 0,Y 331.817,Z 457.352,A -85,B 0,C 180,E1 -15181.883,E2 -15181.883} C_VEL
LIN {X 0,Y 328.046,Z 470.358,A -85,B 0,C 180,E1 -15184.288,E2 -15184.288} C_VEL
LIN {X 0,Y 324.99,Z 481.546,A -85,B 0,C 180,E1 -15186.754,E2 -15186.754} C_VEL
LIN {X 0,Y 322.538,Z 491.14,A -85,B 0,C 180,E1 -15189.262,E2 -15189.262} C_VEL
LIN {X 0,Y 320.485,Z 500.277,A -85,B 0,C 180,E1 -15192.12,E2 -15192.12} C_VEL
LIN {X 0,Y 319.248,Z 507.062,A -85,B 0,C 180,E1 -15194.682,E2 -15194.682} C_VEL
LIN {X 0,Y 318.453,Z 512.581,A -85,B 0,C 180,E1 -15197.25,E2 -15197.25} C_VEL
LIN {X 0,Y 317.996,Z 516.977,A -85,B 0,C 180,E1 -15199.815,E2 -15199.815} C_VEL
LIN {X 0,Y 318.019,Z 520.268,A -85,B 0,C 180,E1 -15202.38,E2 -15202.38} C_VEL
LIN {X 0,Y 318.093,Z 522.416,A -85,B 0,C 180,E1 -15204.929,E2 -15204.929} C_VEL
LIN {X 0,Y 318.254,Z 523.509,A -85,B 0,C 180,E1 -15207.468,E2 -15207.468} C_VEL
LIN {X 0,Y 318.405,Z 523.391,A -85,B 0,C 180,E1 -15209.999,E2 -15209.999} C_VEL
LIN {X 0,Y 318.34,Z 522.177,A -85,B 0,C 180,E1 -15212.53,E2 -15212.53} C_VEL
LIN {X 0,Y 318.2,Z 519.698,A -85,B 0,C 180,E1 -15215.068,E2 -15215.068} C_VEL
LIN {X 0,Y 318.292,Z 517.825,A -85,B 0,C 180,E1 -15216.481,E2 -15216.481} C_VEL
LIN {X 0,Y 318.173,Z 513.73,A -85,B 0,C 180,E1 -15218.894,E2 -15218.894} C_VEL
LIN {X 0,Y 318.311,Z 508.08,A -85,B 0,C 180,E1 -15221.461,E2 -15221.461} C_VEL
LIN {X 0,Y 318.789,Z 500.883,A -85,B 0,C 180,E1 -15224.066,E2 -15224.066} C_VEL
LIN {X 0,Y 319.586,Z 492.313,A -85,B 0,C 180,E1 -15226.611,E2 -15226.611} C_VEL
LIN {X 0,Y 320.709,Z 481.825,A -85,B 0,C 180,E1 -15229.189,E2 -15229.189} C_VEL
LIN {X 0,Y 322.194,Z 470.963,A -85,B 0,C 180,E1 -15231.429,E2 -15231.429} C_VEL
LIN {X 0,Y 323.73,Z 460.126,A -85,B 0,C 180,E1 -15233.34,E2 -15233.34} C_VEL
LIN {X 0,Y 325.636,Z 447.089,A -85,B 0,C 180,E1 -15235.291,E2 -15235.291} C_VEL
LIN {X 0,Y 327.522,Z 433.985,A -85,B 0,C 180,E1 -15236.955,E2 -15236.955} C_VEL
LIN {X 0,Y 329.821,Z 418.025,A -85,B 0,C 180,E1 -15238.648,E2 -15238.648} C_VEL
LIN {X 0,Y 331.903,Z 402.39,A -85,B 0,C 180,E1 -15240.009,E2 -15240.009} C_VEL
LIN {X 0,Y 333.944,Z 385.196,A -85,B 0,C 180,E1 -15241.214,E2 -15241.214} C_VEL
LIN {X 0,Y 335.753,Z 367.466,A -85,B 0,C 180,E1 -15242.171,E2 -15242.171} C_VEL
LIN {X 0,Y 337.222,Z 350.111,A -85,B 0,C 180,E1 -15242.854,E2 -15242.854} C_VEL
LIN {X 0,Y 345.794,Z 198.717,A -85,B 0,C 180,E1 -15247.223,E2 -15247.223} C_VEL
LIN {X 0,Y 343.412,Z 177.184,A -85,B 0,C 180,E1 -15248.167,E2 -15248.167} C_VEL
LIN {X 0,Y 329.969,Z 147.004,A -85,B 0,C 180,E1 -15250.529,E2 -15250.529} C_VEL
LIN {X 0,Y 328.461,Z 143.713,A -85,B 0,C 180,E1 -15250.808,E2 -15250.808} C_VEL
LIN {X 0,Y 322.699,Z 126.126,A -85,B 0,C 180,E1 -15254.053,E2 -15254.053} C_VEL
LIN {X 0,Y 319.547,Z 116.994,A -85,B 0,C 180,E1 -15255.872,E2 -15255.872} C_VEL
LIN {X 0,Y 319.525,Z 116.997,A -85,B 0,C 180,E1 -15258.711,E2 -15258.711} C_VEL
LIN {X 0,Y 319.574,Z 116.992,A -85,B 0,C 180,E1 -15262.344,E2 -15262.344} C_VEL
LIN {X 0,Y 319.556,Z 116.99,A -85,B 0,C 180,E1 -15265.123,E2 -15265.123} C_VEL
LIN {X 0,Y 319.57,Z 116.988,A -85,B 0,C 180,E1 -15269.056,E2 -15269.056} C_VEL
LIN {X 0,Y 319.604,Z 116.986,A -85,B 0,C 180,E1 -15272.498,E2 -15272.498} C_VEL
LIN {X 0,Y 319.6,Z 116.985,A -85,B 0,C 180,E1 -15275.304,E2 -15275.304} C_VEL
LIN {X 0,Y 319.592,Z 116.991,A -85,B 0,C 180,E1 -15278.048,E2 -15278.048} C_VEL
LIN {X 0,Y 319.684,Z 116.974,A -85,B 0,C 180,E1 -15280.962,E2 -15280.962} C_VEL
LIN {X 0,Y 319.726,Z 116.969,A -85,B 0,C 180,E1 -15285.276,E2 -15285.276} C_VEL
LIN {X 0,Y 319.755,Z 116.97,A -85,B 0,C 180,E1 -15289.873,E2 -15289.873} C_VEL
LIN {X 0,Y 319.929,Z 116.943,A -85,B 0,C 180,E1 -15292.426,E2 -15292.426} C_VEL
LIN {X 0,Y 319.744,Z 116.964,A -85,B 0,C 180,E1 -15294.956,E2 -15294.956} C_VEL
LIN {X 0,Y 319.987,Z 116.939,A -85,B 0,C 180,E1 -15297.483,E2 -15297.483} C_VEL
LIN {X 0,Y 320.164,Z 116.916,A -85,B 0,C 180,E1 -15300,E2 -15300} C_VEL
LIN {X 0,Y 319.987,Z 116.935,A -85,B 0,C 180,E1 -15302.518,E2 -15302.518} C_VEL
LIN {X 0,Y 319.927,Z 116.942,A -85,B 0,C 180,E1 -15306.656,E2 -15306.656} C_VEL
LIN {X 0,Y 319.753,Z 116.965,A -85,B 0,C 180,E1 -15310.127,E2 -15310.127} C_VEL
LIN {X 0,Y 319.726,Z 116.969,A -85,B 0,C 180,E1 -15314.725,E2 -15314.725} C_VEL
LIN {X 0,Y 319.684,Z 116.976,A -85,B 0,C 180,E1 -15319.038,E2 -15319.038} C_VEL
LIN {X 0,Y 319.566,Z 116.992,A -85,B 0,C 180,E1 -15323.32,E2 -15323.32} C_VEL
LIN {X 0,Y 319.614,Z 116.982,A -85,B 0,C 180,E1 -15326.09,E2 -15326.09} C_VEL
LIN {X 0,Y 319.576,Z 116.99,A -85,B 0,C 180,E1 -15328.935,E2 -15328.935} C_VEL
LIN {X 0,Y 319.526,Z 116.992,A -85,B 0,C 180,E1 -15331.862,E2 -15331.862} C_VEL
LIN {X 0,Y 319.576,Z 116.988,A -85,B 0,C 180,E1 -15335.544,E2 -15335.544} C_VEL
LIN {X 0,Y 319.555,Z 116.989,A -85,B 0,C 180,E1 -15339.669,E2 -15339.669} C_VEL
LIN {X 0,Y 319.554,Z 116.99,A -85,B 0,C 180,E1 -15343.468,E2 -15343.468} C_VEL
LIN {X 0,Y 319.585,Z 116.988,A -85,B 0,C 180,E1 -15347.023,E2 -15347.023} C_VEL
LIN {X 0,Y 319.579,Z 116.989,A -85,B 0,C 180,E1 -15350.377,E2 -15350.377} C_VEL
LIN {X 0,Y 319.557,Z 116.988,A -85,B 0,C 180,E1 -15353.573,E2 -15353.573} C_VEL
LIN {X 0,Y 319.575,Z 116.992,A -85,B 0,C 180,E1 -15356.687,E2 -15356.687} C_VEL
LIN {X 0,Y 319.582,Z 116.986,A -85,B 0,C 180,E1 -15359.617,E2 -15359.617} C_VEL
LIN {X 0,Y 319.604,Z 116.987,A -85,B 0,C 180,E1 -15362.499,E2 -15362.499} C_VEL
LIN {X 0,Y 319.604,Z 116.983,A -85,B 0,C 180,E1 -15365.305,E2 -15365.305} C_VEL
LIN {X 0,Y 319.621,Z 116.98,A -85,B 0,C 180,E1 -15369.402,E2 -15369.402} C_VEL
LIN {X 0,Y 319.658,Z 116.979,A -85,B 0,C 180,E1 -15372.074,E2 -15372.074} C_VEL
LIN {X 0,Y 319.732,Z 116.969,A -85,B 0,C 180,E1 -15376.009,E2 -15376.009} C_VEL
LIN {X 0,Y 319.758,Z 116.966,A -85,B 0,C 180,E1 -15379.874,E2 -15379.874} C_VEL
LIN {X 0,Y 319.934,Z 116.946,A -85,B 0,C 180,E1 -15382.427,E2 -15382.427} C_VEL
LIN {X 0,Y 319.747,Z 116.965,A -85,B 0,C 180,E1 -15384.957,E2 -15384.957} C_VEL
LIN {X 0,Y 319.99,Z 116.935,A -85,B 0,C 180,E1 -15387.483,E2 -15387.483} C_VEL
LIN {X 0,Y 320.15,Z 116.92,A -85,B 0,C 180,E1 -15390.001,E2 -15390.001} C_VEL
LIN {X 0,Y 319.991,Z 116.935,A -85,B 0,C 180,E1 -15392.518,E2 -15392.518} C_VEL
LIN {X 0,Y 319.953,Z 116.942,A -85,B 0,C 180,E1 -15396.306,E2 -15396.306} C_VEL
LIN {X 0,Y 319.844,Z 116.954,A -85,B 0,C 180,E1 -15398.849,E2 -15398.849} C_VEL
LIN {X 0,Y 319.683,Z 116.973,A -85,B 0,C 180,E1 -15402.701,E2 -15402.701} C_VEL
LIN {X 0,Y 319.701,Z 116.973,A -85,B 0,C 180,E1 -15405.296,E2 -15405.296} C_VEL
LIN {X 0,Y 319.676,Z 116.975,A -85,B 0,C 180,E1 -15409.256,E2 -15409.256} C_VEL
LIN {X 0,Y 319.573,Z 116.989,A -85,B 0,C 180,E1 -15413.32,E2 -15413.32} C_VEL
LIN {X 0,Y 319.636,Z 116.981,A -85,B 0,C 180,E1 -15416.089,E2 -15416.089} C_VEL
LIN {X 0,Y 319.582,Z 116.987,A -85,B 0,C 180,E1 -15418.935,E2 -15418.935} C_VEL
LIN {X 0,Y 319.533,Z 116.995,A -85,B 0,C 180,E1 -15421.863,E2 -15421.863} C_VEL
LIN {X 0,Y 319.583,Z 116.991,A -85,B 0,C 180,E1 -15425.544,E2 -15425.544} C_VEL
LIN {X 0,Y 319.576,Z 116.988,A -85,B 0,C 180,E1 -15428.008,E2 -15428.008} C_VEL
LIN {X 0,Y 319.529,Z 116.996,A -85,B 0,C 180,E1 -15431.598,E2 -15431.598} C_VEL
LIN {X 0,Y 319.519,Z 116.999,A -85,B 0,C 180,E1 -15435.263,E2 -15435.263} C_VEL
LIN {X 0,Y 319.532,Z 116.995,A -85,B 0,C 180,E1 -15438.712,E2 -15438.712} C_VEL
LIN {X 0,Y 319.563,Z 116.993,A -85,B 0,C 180,E1 -15439.352,E2 -15439.352} C_VEL
LIN {X 0,Y 320.553,Z 119.818,A -85,B 0,C 180,E1 -15439.576,E2 -15439.576} C_VEL
LIN {X 0,Y 335.046,Z 147.73,A -85,B 0,C 180,E1 -15442.046,E2 -15442.046} C_VEL
LIN {X 0,Y 344.864,Z 167.675,A -85,B 0,C 180,E1 -15443.62,E2 -15443.62} C_VEL
LIN {X 0,Y 339.65,Z 260.244,A -85,B 0,C 180,E1 -15446.268,E2 -15446.268} C_VEL
LIN {X 0,Y 338.673,Z 266.036,A -85,B 0,C 180,E1 -15446.382,E2 -15446.382} C_VEL
LIN {X 0,Y 332.451,Z 284.84,A -85,B 0,C 180,E1 -15446.546,E2 -15446.546} C_VEL
LIN {X 0,Y 331.473,Z 290.627,A -85,B 0,C 180,E1 -15446.67,E2 -15446.67} C_VEL
LIN {X 0,Y 330.339,Z 309.607,A -85,B 0,C 180,E1 -15447.326,E2 -15447.326} C_VEL
LIN {X 0,Y 329.062,Z 327.108,A -85,B 0,C 180,E1 -15448.179,E2 -15448.179} C_VEL
LIN {X 0,Y 327.515,Z 343.711,A -85,B 0,C 180,E1 -15449.23,E2 -15449.23} C_VEL
LIN {X 0,Y 325.676,Z 360.885,A -85,B 0,C 180,E1 -15450.598,E2 -15450.598} C_VEL
LIN {X 0,Y 323.647,Z 376.97,A -85,B 0,C 180,E1 -15452.168,E2 -15452.168} C_VEL
LIN {X 0,Y 321.621,Z 391.41,A -85,B 0,C 180,E1 -15453.861,E2 -15453.861} C_VEL
LIN {X 0,Y 319.581,Z 405.44,A -85,B 0,C 180,E1 -15455.821,E2 -15455.821} C_VEL
LIN {X 0,Y 317.69,Z 418.078,A -85,B 0,C 180,E1 -15457.909,E2 -15457.909} C_VEL
LIN {X 0,Y 316.089,Z 429.694,A -85,B 0,C 180,E1 -15460.18,E2 -15460.18} C_VEL
LIN {X 0,Y 314.448,Z 440.84,A -85,B 0,C 180,E1 -15462.774,E2 -15462.774} C_VEL
LIN {X 0,Y 313.302,Z 450.18,A -85,B 0,C 180,E1 -15465.399,E2 -15465.399} C_VEL
LIN {X 0,Y 312.46,Z 456.903,A -85,B 0,C 180,E1 -15467.662,E2 -15467.662} C_VEL
LIN {X 0,Y 311.874,Z 463.385,A -85,B 0,C 180,E1 -15470.27,E2 -15470.27} C_VEL
LIN {X 0,Y 311.493,Z 468.974,A -85,B 0,C 180,E1 -15473.098,E2 -15473.098} C_VEL
LIN {X 0,Y 311.239,Z 473.372,A -85,B 0,C 180,E1 -15476.116,E2 -15476.116} C_VEL
LIN {X 0,Y 311.248,Z 475.921,A -85,B 0,C 180,E1 -15478.706,E2 -15478.706} C_VEL
LIN {X 0,Y 311.348,Z 477.501,A -85,B 0,C 180,E1 -15481.293,E2 -15481.293} C_VEL
LIN {X 0,Y 311.711,Z 477.982,A -85,B 0,C 180,E1 -15483.878,E2 -15483.878} C_VEL
LIN {X 0,Y 312.049,Z 477.497,A -85,B 0,C 180,E1 -15486.466,E2 -15486.466} C_VEL
LIN {X 0,Y 312.893,Z 475.981,A -85,B 0,C 180,E1 -15489.046,E2 -15489.046} C_VEL
LIN {X 0,Y 313.939,Z 473.43,A -85,B 0,C 180,E1 -15491.623,E2 -15491.623} C_VEL
LIN {X 0,Y 315.358,Z 469.903,A -85,B 0,C 180,E1 -15494.19,E2 -15494.19} C_VEL
LIN {X 0,Y 317.694,Z 463.912,A -85,B 0,C 180,E1 -15497.376,E2 -15497.376} C_VEL
LIN {X 0,Y 320.815,Z 456.067,A -85,B 0,C 180,E1 -15500.518,E2 -15500.518} C_VEL
LIN {X 0,Y 323.863,Z 448.377,A -85,B 0,C 180,E1 -15502.992,E2 -15502.992} C_VEL
LIN {X 0,Y 327.905,Z 438.113,A -85,B 0,C 180,E1 -15505.688,E2 -15505.688} C_VEL
LIN {X 0,Y 332.08,Z 427.03,A -85,B 0,C 180,E1 -15508.092,E2 -15508.092} C_VEL
LIN {X 0,Y 336.236,Z 415.813,A -85,B 0,C 180,E1 -15510.109,E2 -15510.109} C_VEL
LIN {X 0,Y 340.973,Z 402.24,A -85,B 0,C 180,E1 -15512.181,E2 -15512.181} C_VEL
LIN {X 0,Y 346.097,Z 386.803,A -85,B 0,C 180,E1 -15514.122,E2 -15514.122} C_VEL
LIN {X 0,Y 350.872,Z 371.529,A -85,B 0,C 180,E1 -15515.688,E2 -15515.688} C_VEL
LIN {X 0,Y 355.271,Z 356.076,A -85,B 0,C 180,E1 -15516.996,E2 -15516.996} C_VEL
LIN {X 0,Y 359.244,Z 340.499,A -85,B 0,C 180,E1 -15518.089,E2 -15518.089} C_VEL
LIN {X 0,Y 363.156,Z 323.07,A -85,B 0,C 180,E1 -15519.062,E2 -15519.062} C_VEL
LIN {X 0,Y 368.505,Z 296.148,A -85,B 0,C 180,E1 -15520.155,E2 -15520.155} C_VEL
LIN {X 0,Y 383.534,Z 229.224,A -85,B 0,C 180,E1 -15522.598,E2 -15522.598} C_VEL
LIN {X 0,Y 388.258,Z 209.929,A -85,B 0,C 180,E1 -15523.298,E2 -15523.298} C_VEL
LIN {X 0,Y 387.796,Z 211.477,A -85,B 0,C 180,E1 -15524.875,E2 -15524.875} C_VEL
LIN {X 0,Y 387.698,Z 213.263,A -85,B 0,C 180,E1 -15525.667,E2 -15525.667} C_VEL
LIN {X 0,Y 376.155,Z 263.605,A -85,B 0,C 180,E1 -15527.458,E2 -15527.458} C_VEL
LIN {X 0,Y 363.544,Z 326.251,A -85,B 0,C 180,E1 -15529.773,E2 -15529.773} C_VEL
LIN {X 0,Y 359.256,Z 346.949,A -85,B 0,C 180,E1 -15530.612,E2 -15530.612} C_VEL
LIN {X 0,Y 354.528,Z 365.716,A -85,B 0,C 180,E1 -15531.54,E2 -15531.54} C_VEL
